LIN {X 0,Y 235.109,Z 274.18,A -85,B 0,C 180,E1 -19787.924,E2 -19787.924} C_VEL
LIN {X 0,Y 235.327,Z 274.163,A -85,B 0,C 180,E1 -19791.414,E2 -19791.414} C_VEL
LIN {X 0,Y 235.369,Z 274.162,A -85,B 0,C 180,E1 -19793.142,E2 -19793.142} C_VEL
LIN {X 0,Y 235.592,Z 274.14,A -85,B 0,C 180,E1 -19798.293,E2 -19798.293} C_VEL
LIN {X 0,Y 235.593,Z 274.134,A -85,B 0,C 180,E1 -19801.711,E2 -19801.711} C_VEL
LIN {X 0,Y 235.402,Z 274.153,A -85,B 0,C 180,E1 -19806.861,E2 -19806.861} C_VEL
LIN {X 0,Y 235.237,Z 274.182,A -85,B 0,C 180,E1 -19810.328,E2 -19810.328} C_VEL
LIN {X 0,Y 235.107,Z 274.198,A -85,B 0,C 180,E1 -19815.609,E2 -19815.609} C_VEL
LIN {X 0,Y 235.007,Z 274.203,A -85,B 0,C 180,E1 -19819.208,E2 -19819.208} C_VEL
LIN {X 0,Y 234.961,Z 274.215,A -85,B 0,C 180,E1 -19822.885,E2 -19822.885} C_VEL
LIN {X 0,Y 234.97,Z 274.212,A -85,B 0,C 180,E1 -19826.659,E2 -19826.659} C_VEL
LIN {X 0,Y 234.933,Z 274.22,A -85,B 0,C 180,E1 -19830.57,E2 -19830.57} C_VEL
LIN {X 0,Y 234.929,Z 274.22,A -85,B 0,C 180,E1 -19834.64,E2 -19834.64} C_VEL
LIN {X 0,Y 234.945,Z 274.221,A -85,B 0,C 180,E1 -19838.946,E2 -19838.946} C_VEL
LIN {X 0,Y 234.971,Z 274.365,A -85,B 0,C 180,E1 -19843.971,E2 -19843.971} C_VEL
LIN {X 0,Y 235.687,Z 278.299,A -85,B 0,C 180,E1 -19848.203,E2 -19848.203} C_VEL
LIN {X 0,Y 236.227,Z 281.355,A -85,B 0,C 180,E1 -19851.335,E2 -19851.335} C_VEL
LIN {X 0,Y 236.327,Z 282.58,A -85,B 0,C 180,E1 -19852.548,E2 -19852.548} C_VEL
LIN {X 0,Y 235.561,Z 284.082,A -85,B 0,C 180,E1 -19853.919,E2 -19853.919} C_VEL
LIN {X 0,Y 233.781,Z 285.659,A -85,B 0,C 180,E1 -19855.25,E2 -19855.25} C_VEL
LIN {X 0,Y 229.483,Z 288.871,A -85,B 0,C 180,E1 -19857.918,E2 -19857.918} C_VEL
LIN {X 0,Y 228.112,Z 290.471,A -85,B 0,C 180,E1 -19859.328,E2 -19859.328} C_VEL
LIN {X 0,Y 227.922,Z 290.995,A -85,B 0,C 180,E1 -19859.811,E2 -19859.811} C_VEL
LIN {X 0,Y 227.643,Z 292.579,A -85,B 0,C 180,E1 -19861.29,E2 -19861.29} C_VEL
LIN {X 0,Y 230.37,Z 306.658,A -85,B 0,C 180,E1 -19862.479,E2 -19862.479} C_VEL
LIN {X 0,Y 232.357,Z 320.143,A -85,B 0,C 180,E1 -19863.933,E2 -19863.933} C_VEL
LIN {X 0,Y 233.562,Z 332.37,A -85,B 0,C 180,E1 -19865.56,E2 -19865.56} C_VEL
LIN {X 0,Y 234.118,Z 342.965,A -85,B 0,C 180,E1 -19867.264,E2 -19867.264} C_VEL
LIN {X 0,Y 232.286,Z 353.457,A -85,B 0,C 180,E1 -19869.176,E2 -19869.176} C_VEL
LIN {X 0,Y 230.426,Z 363.523,A -85,B 0,C 180,E1 -19871.471,E2 -19871.471} C_VEL
LIN {X 0,Y 228.848,Z 372.161,A -85,B 0,C 180,E1 -19873.955,E2 -19873.955} C_VEL
LIN {X 0,Y 227.39,Z 379.539,A -85,B 0,C 180,E1 -19876.597,E2 -19876.597} C_VEL
LIN {X 0,Y 226.524,Z 385.469,A -85,B 0,C 180,E1 -19879.272,E2 -19879.272} C_VEL
LIN {X 0,Y 225.961,Z 390.122,A -85,B 0,C 180,E1 -19881.954,E2 -19881.954} C_VEL
LIN {X 0,Y 225.657,Z 393.634,A -85,B 0,C 180,E1 -19884.639,E2 -19884.639} C_VEL
LIN {X 0,Y 225.627,Z 395.395,A -85,B 0,C 180,E1 -19886.428,E2 -19886.428} C_VEL
LIN {X 0,Y 225.692,Z 396.715,A -85,B 0,C 180,E1 -19888.215,E2 -19888.215} C_VEL
LIN {X 0,Y 225.758,Z 397.627,A -85,B 0,C 180,E1 -19890,E2 -19890} C_VEL
LIN {X 0,Y 225.659,Z 398.135,A -85,B 0,C 180,E1 -19891.784,E2 -19891.784} C_VEL
LIN {X 0,Y 225.601,Z 398.096,A -85,B 0,C 180,E1 -19894.512,E2 -19894.512} C_VEL
LIN {X 0,Y 225.831,Z 397.183,A -85,B 0,C 180,E1 -19897.15,E2 -19897.15} C_VEL
LIN {X 0,Y 226.166,Z 396.101,A -85,B 0,C 180,E1 -19898.938,E2 -19898.938} C_VEL
LIN {X 0,Y 226.673,Z 394.603,A -85,B 0,C 180,E1 -19900.721,E2 -19900.721} C_VEL
LIN {X 0,Y 227.781,Z 391.576,A -85,B 0,C 180,E1 -19903.379,E2 -19903.379} C_VEL
LIN {X 0,Y 229.362,Z 387.538,A -85,B 0,C 180,E1 -19906.008,E2 -19906.008} C_VEL
LIN {X 0,Y 231.967,Z 381.395,A -85,B 0,C 180,E1 -19909.007,E2 -19909.007} C_VEL
LIN {X 0,Y 234.464,Z 374.434,A -85,B 0,C 180,E1 -19911.683,E2 -19911.683} C_VEL
LIN {X 0,Y 237.395,Z 366.72,A -85,B 0,C 180,E1 -19914.02,E2 -19914.02} C_VEL
LIN {X 0,Y 240.409,Z 358.529,A -85,B 0,C 180,E1 -19916.007,E2 -19916.007} C_VEL
LIN {X 0,Y 242.378,Z 352.8,A -85,B 0,C 180,E1 -19917.173,E2 -19917.173} C_VEL
LIN {X 0,Y 243.214,Z 343.096,A -85,B 0,C 180,E1 -19919.215,E2 -19919.215} C_VEL
LIN {X 0,Y 242.953,Z 333.446,A -85,B 0,C 180,E1 -19921.135,E2 -19921.135} C_VEL
LIN {X 0,Y 241.554,Z 322.509,A -85,B 0,C 180,E1 -19923.227,E2 -19923.227} C_VEL
LIN {X 0,Y 238.999,Z 311.749,A -85,B 0,C 180,E1 -19925.301,E2 -19925.301} C_VEL
LIN {X 0,Y 235.898,Z 302.595,A -85,B 0,C 180,E1 -19927.162,E2 -19927.162} C_VEL
LIN {X 0,Y 234.604,Z 299.647,A -85,B 0,C 180,E1 -19927.81,E2 -19927.81} C_VEL
LIN {X 0,Y 232.641,Z 295.3,A -85,B 0,C 180,E1 -19928.793,E2 -19928.793} C_VEL
LIN {X 0,Y 230.868,Z 292.3,A -85,B 0,C 180,E1 -19929.608,E2 -19929.608} C_VEL
LIN {X 0,Y 230.247,Z 290.185,A -85,B 0,C 180,E1 -19930.007,E2 -19930.007} C_VEL
LIN {X 0,Y 230.039,Z 288.162,A -85,B 0,C 180,E1 -19932.839,E2 -19932.839} C_VEL
LIN {X 0,Y 229.659,Z 285.357,A -85,B 0,C 180,E1 -19937.259,E2 -19937.259} C_VEL
LIN {X 0,Y 229.411,Z 283.843,A -85,B 0,C 180,E1 -19939.983,E2 -19939.983} C_VEL
LIN {X 0,Y 229.062,Z 281.787,A -85,B 0,C 180,E1 -19944.339,E2 -19944.339} C_VEL
LIN {X 0,Y 228.798,Z 280.217,A -85,B 0,C 180,E1 -19948.519,E2 -19948.519} C_VEL
LIN {X 0,Y 228.652,Z 278.956,A -85,B 0,C 180,E1 -19953.042,E2 -19953.042} C_VEL
LIN {X 0,Y 228.5,Z 278.111,A -85,B 0,C 180,E1 -19958.339,E2 -19958.339} C_VEL
LIN {X 0,Y 228.515,Z 277.888,A -85,B 0,C 180,E1 -19962.437,E2 -19962.437} C_VEL
LIN {X 0,Y 228.587,Z 277.979,A -85,B 0,C 180,E1 -19965.759,E2 -19965.759} C_VEL
LIN {X 0,Y 228.79,Z 278.339,A -85,B 0,C 180,E1 -19969.407,E2 -19969.407} C_VEL
LIN {X 0,Y 228.966,Z 278.971,A -85,B 0,C 180,E1 -19972.946,E2 -19972.946} C_VEL
LIN {X 0,Y 229.425,Z 280.374,A -85,B 0,C 180,E1 -19978.243,E2 -19978.243} C_VEL
LIN {X 0,Y 229.645,Z 280.948,A -85,B 0,C 180,E1 -19979.998,E2 -19979.998} C_VEL
LIN {X 0,Y 229.49,Z 282.382,A -85,B 0,C 180,E1 -19983.509,E2 -19983.509} C_VEL
LIN {X 0,Y 229.473,Z 283.455,A -85,B 0,C 180,E1 -19985.876,E2 -19985.876} C_VEL
LIN {X 0,Y 230.504,Z 286.209,A -85,B 0,C 180,E1 -19986.453,E2 -19986.453} C_VEL
LIN {X 0,Y 232.638,Z 289.092,A -85,B 0,C 180,E1 -19987.388,E2 -19987.388} C_VEL
LIN {X 0,Y 234.347,Z 292.521,A -85,B 0,C 180,E1 -19988.256,E2 -19988.256} C_VEL
LIN {X 0,Y 238.089,Z 300.635,A -85,B 0,C 180,E1 -19990.199,E2 -19990.199} C_VEL
LIN {X 0,Y 241.76,Z 311.494,A -85,B 0,C 180,E1 -19992.608,E2 -19992.608} C_VEL
LIN {X 0,Y 243.899,Z 320.884,A -85,B 0,C 180,E1 -19994.602,E2 -19994.602} C_VEL
LIN {X 0,Y 245.093,Z 330.377,A -85,B 0,C 180,E1 -19996.661,E2 -19996.661} C_VEL
LIN {X 0,Y 245.285,Z 336.573,A -85,B 0,C 180,E1 -19998.035,E2 -19998.035} C_VEL
LIN {X 0,Y 242.242,Z 346.347,A -85,B 0,C 180,E1 -19999.929,E2 -19999.929} C_VEL
LIN {X 0,Y 239.08,Z 355.259,A -85,B 0,C 180,E1 -20002.077,E2 -20002.077} C_VEL
LIN {X 0,Y 235.802,Z 363.65,A -85,B 0,C 180,E1 -20004.66,E2 -20004.66} C_VEL
LIN {X 0,Y 233.456,Z 369.311,A -85,B 0,C 180,E1 -20006.841,E2 -20006.841} C_VEL
LIN {X 0,Y 231.392,Z 374.044,A -85,B 0,C 180,E1 -20009.073,E2 -20009.073} C_VEL
LIN {X 0,Y 229.708,Z 377.876,A -85,B 0,C 180,E1 -20011.338,E2 -20011.338} C_VEL
LIN {X 0,Y 227.769,Z 382.127,A -85,B 0,C 180,E1 -20014.809,E2 -20014.809} C_VEL
LIN {X 0,Y 226.387,Z 384.802,A -85,B 0,C 180,E1 -20018.378,E2 -20018.378} C_VEL
LIN {X 0,Y 225.615,Z 385.794,A -85,B 0,C 180,E1 -20021.618,E2 -20021.618} C_VEL
LIN {X 0,Y 225.292,Z 385.696,A -85,B 0,C 180,E1 -20024.154,E2 -20024.154} C_VEL
LIN {X 0,Y 225.213,Z 384.787,A -85,B 0,C 180,E1 -20026.645,E2 -20026.645} C_VEL
LIN {X 0,Y 225.305,Z 383.158,A -85,B 0,C 180,E1 -20029.077,E2 -20029.077} C_VEL
LIN {X 0,Y 225.669,Z 380.804,A -85,B 0,C 180,E1 -20031.476,E2 -20031.476} C_VEL
LIN {X 0,Y 226.183,Z 377.61,A -85,B 0,C 180,E1 -20033.885,E2 -20033.885} C_VEL
LIN {X 0,Y 226.991,Z 372.694,A -85,B 0,C 180,E1 -20036.712,E2 -20036.712} C_VEL
LIN {X 0,Y 228.158,Z 366.18,A -85,B 0,C 180,E1 -20039.592,E2 -20039.592} C_VEL
LIN {X 0,Y 229.753,Z 357.785,A -85,B 0,C 180,E1 -20042.504,E2 -20042.504} C_VEL
LIN {X 0,Y 231.376,Z 349.279,A -85,B 0,C 180,E1 -20044.834,E2 -20044.834} C_VEL
LIN {X 0,Y 233.076,Z 339.892,A -85,B 0,C 180,E1 -20046.922,E2 -20046.922} C_VEL
LIN {X 0,Y 234.817,Z 330.283,A -85,B 0,C 180,E1 -20048.654,E2 -20048.654} C_VEL
LIN {X 0,Y 235.628,Z 324.925,A -85,B 0,C 180,E1 -20049.485,E2 -20049.485} C_VEL
LIN {X 0,Y 234.384,Z 314.919,A -85,B 0,C 180,E1 -20051.017,E2 -20051.017} C_VEL
LIN {X 0,Y 232.292,Z 302.871,A -85,B 0,C 180,E1 -20052.582,E2 -20052.582} C_VEL
LIN {X 0,Y 229.337,Z 289.586,A -85,B 0,C 180,E1 -20053.991,E2 -20053.991} C_VEL
LIN {X 0,Y 227.152,Z 280.91,A -85,B 0,C 180,E1 -20054.753,E2 -20054.753} C_VEL
LIN {X 0,Y 227.624,Z 277.181,A -85,B 0,C 180,E1 -20059.325,E2 -20059.325} C_VEL
LIN {X 0,Y 228.142,Z 275.067,A -85,B 0,C 180,E1 -20062.032,E2 -20062.032} C_VEL
LIN {X 0,Y 228.544,Z 275.016,A -85,B 0,C 180,E1 -20068.238,E2 -20068.238} C_VEL
LIN {X 0,Y 228.548,Z 275.015,A -85,B 0,C 180,E1 -20071.762,E2 -20071.762} C_VEL
LIN {X 0,Y 228.349,Z 275.041,A -85,B 0,C 180,E1 -20077.072,E2 -20077.072} C_VEL
LIN {X 0,Y 228.163,Z 275.062,A -85,B 0,C 180,E1 -20080.65,E2 -20080.65} C_VEL
LIN {X 0,Y 228.049,Z 275.077,A -85,B 0,C 180,E1 -20086.103,E2 -20086.103} C_VEL
LIN {X 0,Y 227.946,Z 275.088,A -85,B 0,C 180,E1 -20089.825,E2 -20089.825} C_VEL
LIN {X 0,Y 227.917,Z 275.095,A -85,B 0,C 180,E1 -20093.632,E2 -20093.632} C_VEL
LIN {X 0,Y 227.871,Z 275.093,A -85,B 0,C 180,E1 -20097.557,E2 -20097.557} C_VEL
LIN {X 0,Y 227.861,Z 275.1,A -85,B 0,C 180,E1 -20101.623,E2 -20101.623} C_VEL
LIN {X 0,Y 227.893,Z 275.097,A -85,B 0,C 180,E1 -20105.869,E2 -20105.869} C_VEL
LIN {X 0,Y 227.896,Z 275.085,A -85,B 0,C 180,E1 -20110.361,E2 -20110.361} C_VEL
LIN {X 0,Y 227.912,Z 275.086,A -85,B 0,C 180,E1 -20114.831,E2 -20114.831} C_VEL
LIN {X 0,Y 227.919,Z 275.093,A -85,B 0,C 180,E1 -20117.735,E2 -20117.735} C_VEL
LIN {X 0,Y 227.864,Z 275.099,A -85,B 0,C 180,E1 -20121.916,E2 -20121.916} C_VEL
LIN {X 0,Y 227.883,Z 275.089,A -85,B 0,C 180,E1 -20126.375,E2 -20126.375} C_VEL
LIN {X 0,Y 227.913,Z 275.078,A -85,B 0,C 180,E1 -20130.44,E2 -20130.44} C_VEL
LIN {X 0,Y 227.923,Z 275.088,A -85,B 0,C 180,E1 -20134.428,E2 -20134.428} C_VEL
LIN {X 0,Y 227.957,Z 275.089,A -85,B 0,C 180,E1 -20138.289,E2 -20138.289} C_VEL
LIN {X 0,Y 228.03,Z 275.076,A -85,B 0,C 180,E1 -20142.828,E2 -20142.828} C_VEL
LIN {X 0,Y 228.067,Z 275.056,A -85,B 0,C 180,E1 -20147.545,E2 -20147.545} C_VEL
LIN {X 0,Y 228.263,Z 275.043,A -85,B 0,C 180,E1 -20151.147,E2 -20151.147} C_VEL
LIN {X 0,Y 228.32,Z 275.041,A -85,B 0,C 180,E1 -20152.93,E2 -20152.93} C_VEL
LIN {X 0,Y 228.551,Z 275.017,A -85,B 0,C 180,E1 -20158.24,E2 -20158.24} C_VEL
LIN {X 0,Y 228.552,Z 275.011,A -85,B 0,C 180,E1 -20161.764,E2 -20161.764} C_VEL
LIN {X 0,Y 228.353,Z 275.031,A -85,B 0,C 180,E1 -20167.074,E2 -20167.074} C_VEL
LIN {X 0,Y 228.162,Z 275.062,A -85,B 0,C 180,E1 -20170.652,E2 -20170.652} C_VEL
LIN {X 0,Y 228.053,Z 275.073,A -85,B 0,C 180,E1 -20176.104,E2 -20176.104} C_VEL
LIN {X 0,Y 227.942,Z 275.086,A -85,B 0,C 180,E1 -20179.828,E2 -20179.828} C_VEL
LIN {X 0,Y 227.915,Z 275.097,A -85,B 0,C 180,E1 -20183.635,E2 -20183.635} C_VEL
LIN {X 0,Y 227.886,Z 275.095,A -85,B 0,C 180,E1 -20187.557,E2 -20187.557} C_VEL
LIN {X 0,Y 227.872,Z 275.103,A -85,B 0,C 180,E1 -20191.624,E2 -20191.624} C_VEL
LIN {X 0,Y 227.882,Z 275.097,A -85,B 0,C 180,E1 -20195.874,E2 -20195.874} C_VEL
LIN {X 0,Y 227.829,Z 275.104,A -85,B 0,C 180,E1 -20200.378,E2 -20200.378} C_VEL
LIN {X 0,Y 227.93,Z 275.125,A -85,B 0,C 180,E1 -20203.626,E2 -20203.626} C_VEL
LIN {X 0,Y 228.53,Z 278.675,A -85,B 0,C 180,E1 -20207.57,E2 -20207.57} C_VEL
LIN {X 0,Y 229.161,Z 282.067,A -85,B 0,C 180,E1 -20211.17,E2 -20211.17} C_VEL
LIN {X 0,Y 229.294,Z 283.707,A -85,B 0,C 180,E1 -20212.839,E2 -20212.839} C_VEL
LIN {X 0,Y 229.191,Z 285.251,A -85,B 0,C 180,E1 -20214.365,E2 -20214.365} C_VEL
LIN {X 0,Y 228.258,Z 289.527,A -85,B 0,C 180,E1 -20218.438,E2 -20218.438} C_VEL
LIN {X 0,Y 227.922,Z 290.995,A -85,B 0,C 180,E1 -20219.811,E2 -20219.811} C_VEL
LIN {X 0,Y 227.69,Z 292.595,A -85,B 0,C 180,E1 -20220.522,E2 -20220.522} C_VEL
LIN {X 0,Y 227.27,Z 296.129,A -85,B 0,C 180,E1 -20221.199,E2 -20221.199} C_VEL
LIN {X 0,Y 226.616,Z 301.709,A -85,B 0,C 180,E1 -20221.731,E2 -20221.731} C_VEL
LIN {X 0,Y 225.166,Z 314.703,A -85,B 0,C 180,E1 -20222.738,E2 -20222.738} C_VEL
LIN {X 0,Y 225.343,Z 319.397,A -85,B 0,C 180,E1 -20223.261,E2 -20223.261} C_VEL
LIN {X 0,Y 226.472,Z 330.659,A -85,B 0,C 180,E1 -20224.786,E2 -20224.786} C_VEL
LIN {X 0,Y 227.246,Z 342.743,A -85,B 0,C 180,E1 -20226.777,E2 -20226.777} C_VEL
LIN {X 0,Y 225.411,Z 353.248,A -85,B 0,C 180,E1 -20228.749,E2 -20228.749} C_VEL
LIN {X 0,Y 223.533,Z 362.941,A -85,B 0,C 180,E1 -20231.011,E2 -20231.011} C_VEL
LIN {X 0,Y 221.938,Z 371.269,A -85,B 0,C 180,E1 -20233.441,E2 -20233.441} C_VEL
LIN {X 0,Y 220.454,Z 378.773,A -85,B 0,C 180,E1 -20236.167,E2 -20236.167} C_VEL
LIN {X 0,Y 219.512,Z 384.809,A -85,B 0,C 180,E1 -20238.925,E2 -20238.925} C_VEL
LIN {X 0,Y 218.904,Z 389.56,A -85,B 0,C 180,E1 -20241.693,E2 -20241.693} C_VEL
LIN {X 0,Y 218.581,Z 393.165,A -85,B 0,C 180,E1 -20244.465,E2 -20244.465} C_VEL
LIN {X 0,Y 218.527,Z 395.006,A -85,B 0,C 180,E1 -20246.312,E2 -20246.312} C_VEL
LIN {X 0,Y 218.606,Z 396.372,A -85,B 0,C 180,E1 -20248.157,E2 -20248.157} C_VEL
LIN {X 0,Y 218.671,Z 397.323,A -85,B 0,C 180,E1 -20250,E2 -20250} C_VEL
LIN {X 0,Y 218.574,Z 397.87,A -85,B 0,C 180,E1 -20251.842,E2 -20251.842} C_VEL
LIN {X 0,Y 218.519,Z 397.943,A -85,B 0,C 180,E1 -20254.403,E2 -20254.403} C_VEL
LIN {X 0,Y 218.77,Z 397.089,A -85,B 0,C 180,E1 -20257.383,E2 -20257.383} C_VEL
LIN {X 0,Y 219.681,Z 394.626,A -85,B 0,C 180,E1 -20261.066,E2 -20261.066} C_VEL
LIN {X 0,Y 220.853,Z 391.671,A -85,B 0,C 180,E1 -20263.807,E2 -20263.807} C_VEL
LIN {X 0,Y 222.561,Z 387.73,A -85,B 0,C 180,E1 -20266.51,E2 -20266.51} C_VEL
LIN {X 0,Y 224.863,Z 382.723,A -85,B 0,C 180,E1 -20269.157,E2 -20269.157} C_VEL
LIN {X 0,Y 227.306,Z 376.526,A -85,B 0,C 180,E1 -20271.778,E2 -20271.778} C_VEL
LIN {X 0,Y 230.379,Z 368.865,A -85,B 0,C 180,E1 -20274.319,E2 -20274.319} C_VEL
LIN {X 0,Y 233.424,Z 361.125,A -85,B 0,C 180,E1 -20276.365,E2 -20276.365} C_VEL
LIN {X 0,Y 236.129,Z 353.835,A -85,B 0,C 180,E1 -20277.954,E2 -20277.954} C_VEL
LIN {X 0,Y 237.12,Z 343.537,A -85,B 0,C 180,E1 -20280.255,E2 -20280.255} C_VEL
LIN {X 0,Y 237.032,Z 335.241,A -85,B 0,C 180,E1 -20282.004,E2 -20282.004} C_VEL
LIN {X 0,Y 235.875,Z 324.703,A -85,B 0,C 180,E1 -20284.157,E2 -20284.157} C_VEL
LIN {X 0,Y 233.34,Z 313.355,A -85,B 0,C 180,E1 -20286.523,E2 -20286.523} C_VEL
LIN {X 0,Y 230.672,Z 305.204,A -85,B 0,C 180,E1 -20288.319,E2 -20288.319} C_VEL
LIN {X 0,Y 228.334,Z 300.11,A -85,B 0,C 180,E1 -20289.624,E2 -20289.624} C_VEL
LIN {X 0,Y 226.59,Z 296.359,A -85,B 0,C 180,E1 -20290.586,E2 -20290.586} C_VEL
LIN {X 0,Y 223.827,Z 292.087,A -85,B 0,C 180,E1 -20291.976,E2 -20291.976} C_VEL
LIN {X 0,Y 223.131,Z 289.834,A -85,B 0,C 180,E1 -20292.466,E2 -20292.466} C_VEL
LIN {X 0,Y 222.765,Z 287.298,A -85,B 0,C 180,E1 -20296.519,E2 -20296.519} C_VEL
LIN {X 0,Y 222.404,Z 285.015,A -85,B 0,C 180,E1 -20300.8,E2 -20300.8} C_VEL
LIN {X 0,Y 222.282,Z 283.94,A -85,B 0,C 180,E1 -20303.075,E2 -20303.075} C_VEL
LIN {X 0,Y 221.909,Z 281.809,A -85,B 0,C 180,E1 -20308.769,E2 -20308.769} C_VEL
LIN {X 0,Y 221.73,Z 280.535,A -85,B 0,C 180,E1 -20313.655,E2 -20313.655} C_VEL
LIN {X 0,Y 221.621,Z 279.903,A -85,B 0,C 180,E1 -20317.631,E2 -20317.631} C_VEL
LIN {X 0,Y 221.618,Z 279.603,A -85,B 0,C 180,E1 -20322.054,E2 -20322.054} C_VEL
LIN {X 0,Y 221.742,Z 279.781,A -85,B 0,C 180,E1 -20327.18,E2 -20327.18} C_VEL
LIN {X 0,Y 221.981,Z 280.226,A -85,B 0,C 180,E1 -20330.89,E2 -20330.89} C_VEL
LIN {X 0,Y 222.095,Z 280.973,A -85,B 0,C 180,E1 -20334.55,E2 -20334.55} C_VEL
LIN {X 0,Y 222.483,Z 281.915,A -85,B 0,C 180,E1 -20338.188,E2 -20338.188} C_VEL
LIN {X 0,Y 222.723,Z 282.485,A -85,B 0,C 180,E1 -20339.998,E2 -20339.998} C_VEL
LIN {X 0,Y 222.565,Z 283.867,A -85,B 0,C 180,E1 -20343.449,E2 -20343.449} C_VEL
LIN {X 0,Y 223.585,Z 286.659,A -85,B 0,C 180,E1 -20344.11,E2 -20344.11} C_VEL
LIN {X 0,Y 225.858,Z 289.561,A -85,B 0,C 180,E1 -20345.244,E2 -20345.244} C_VEL
LIN {X 0,Y 227.79,Z 293.241,A -85,B 0,C 180,E1 -20346.308,E2 -20346.308} C_VEL
LIN {X 0,Y 228.833,Z 294.901,A -85,B 0,C 180,E1 -20346.833,E2 -20346.833} C_VEL
LIN {X 0,Y 232.06,Z 301.788,A -85,B 0,C 180,E1 -20348.707,E2 -20348.707} C_VEL
LIN {X 0,Y 235.597,Z 311.998,A -85,B 0,C 180,E1 -20351.178,E2 -20351.178} C_VEL
LIN {X 0,Y 237.724,Z 321.242,A -85,B 0,C 180,E1 -20353.309,E2 -20353.309} C_VEL
LIN {X 0,Y 238.91,Z 330.177,A -85,B 0,C 180,E1 -20355.35,E2 -20355.35} C_VEL
LIN {X 0,Y 239.149,Z 337.532,A -85,B 0,C 180,E1 -20357.088,E2 -20357.088} C_VEL
LIN {X 0,Y 238.37,Z 340.868,A -85,B 0,C 180,E1 -20357.768,E2 -20357.768} C_VEL
LIN {X 0,Y 234.671,Z 351.265,A -85,B 0,C 180,E1 -20360.027,E2 -20360.027} C_VEL
LIN {X 0,Y 231.462,Z 359.483,A -85,B 0,C 180,E1 -20362.303,E2 -20362.303} C_VEL
LIN {X 0,Y 228.097,Z 367.313,A -85,B 0,C 180,E1 -20365.063,E2 -20365.063} C_VEL
LIN {X 0,Y 225.244,Z 373.544,A -85,B 0,C 180,E1 -20367.904,E2 -20367.904} C_VEL
LIN {X 0,Y 223.335,Z 377.492,A -85,B 0,C 180,E1 -20370.229,E2 -20370.229} C_VEL
LIN {X 0,Y 221.811,Z 380.64,A -85,B 0,C 180,E1 -20372.588,E2 -20372.588} C_VEL
LIN {X 0,Y 220.572,Z 383.083,A -85,B 0,C 180,E1 -20374.993,E2 -20374.993} C_VEL
LIN {X 0,Y 219.566,Z 384.776,A -85,B 0,C 180,E1 -20377.454,E2 -20377.454} C_VEL
LIN {X 0,Y 218.858,Z 385.772,A -85,B 0,C 180,E1 -20379.956,E2 -20379.956} C_VEL
LIN {X 0,Y 218.37,Z 386.06,A -85,B 0,C 180,E1 -20382.518,E2 -20382.518} C_VEL
LIN {X 0,Y 218.151,Z 385.546,A -85,B 0,C 180,E1 -20385.13,E2 -20385.13} C_VEL
LIN {X 0,Y 218.13,Z 384.183,A -85,B 0,C 180,E1 -20387.817,E2 -20387.817} C_VEL
LIN {X 0,Y 218.392,Z 381.901,A -85,B 0,C 180,E1 -20390.56,E2 -20390.56} C_VEL
LIN {X 0,Y 218.947,Z 378.567,A -85,B 0,C 180,E1 -20393.363,E2 -20393.363} C_VEL
LIN {X 0,Y 219.736,Z 373.943,A -85,B 0,C 180,E1 -20396.257,E2 -20396.257} C_VEL
LIN {X 0,Y 220.932,Z 367.358,A -85,B 0,C 180,E1 -20399.406,E2 -20399.406} C_VEL
LIN {X 0,Y 222.428,Z 359.779,A -85,B 0,C 180,E1 -20402.21,E2 -20402.21} C_VEL
LIN {X 0,Y 223.972,Z 351.723,A -85,B 0,C 180,E1 -20404.613,E2 -20404.613} C_VEL
LIN {X 0,Y 225.748,Z 342.461,A -85,B 0,C 180,E1 -20406.857,E2 -20406.857} C_VEL
LIN {X 0,Y 227.81,Z 331.358,A -85,B 0,C 180,E1 -20408.984,E2 -20408.984} C_VEL
LIN {X 0,Y 228.744,Z 324.991,A -85,B 0,C 180,E1 -20410.014,E2 -20410.014} C_VEL
LIN {X 0,Y 227.271,Z 313.977,A -85,B 0,C 180,E1 -20411.755,E2 -20411.755} C_VEL
LIN {X 0,Y 225.176,Z 302.364,A -85,B 0,C 180,E1 -20413.291,E2 -20413.291} C_VEL
LIN {X 0,Y 222.114,Z 288.88,A -85,B 0,C 180,E1 -20414.751,E2 -20414.751} C_VEL
LIN {X 0,Y 220.157,Z 281.048,A -85,B 0,C 180,E1 -20415.5,E2 -20415.5} C_VEL
LIN {X 0,Y 221.033,Z 276.124,A -85,B 0,C 180,E1 -20421.774,E2 -20421.774} C_VEL
LIN {X 0,Y 221.091,Z 275.944,A -85,B 0,C 180,E1 -20424.528,E2 -20424.528} C_VEL
LIN {X 0,Y 221.501,Z 275.893,A -85,B 0,C 180,E1 -20428.182,E2 -20428.182} C_VEL
LIN {X 0,Y 221.506,Z 275.892,A -85,B 0,C 180,E1 -20431.818,E2 -20431.818} C_VEL
LIN {X 0,Y 221.302,Z 275.919,A -85,B 0,C 180,E1 -20437.298,E2 -20437.298} C_VEL
LIN {X 0,Y 221.108,Z 275.939,A -85,B 0,C 180,E1 -20440.994,E2 -20440.994} C_VEL
LIN {X 0,Y 221.008,Z 275.951,A -85,B 0,C 180,E1 -20446.63,E2 -20446.63} C_VEL
LIN {X 0,Y 220.901,Z 275.968,A -85,B 0,C 180,E1 -20450.485,E2 -20450.485} C_VEL
LIN {X 0,Y 220.865,Z 275.97,A -85,B 0,C 180,E1 -20454.435,E2 -20454.435} C_VEL
LIN {X 0,Y 220.818,Z 275.969,A -85,B 0,C 180,E1 -20458.516,E2 -20458.516} C_VEL
LIN {X 0,Y 220.815,Z 275.977,A -85,B 0,C 180,E1 -20462.756,E2 -20462.756} C_VEL
LIN {X 0,Y 220.83,Z 275.976,A -85,B 0,C 180,E1 -20467.289,E2 -20467.289} C_VEL
LIN {X 0,Y 220.866,Z 275.957,A -85,B 0,C 180,E1 -20471.93,E2 -20471.93} C_VEL
LIN {X 0,Y 220.866,Z 275.969,A -85,B 0,C 180,E1 -20475.573,E2 -20475.573} C_VEL
LIN {X 0,Y 220.851,Z 275.974,A -85,B 0,C 180,E1 -20479.794,E2 -20479.794} C_VEL
LIN {X 0,Y 220.828,Z 275.976,A -85,B 0,C 180,E1 -20482.797,E2 -20482.797} C_VEL
LIN {X 0,Y 220.817,Z 275.964,A -85,B 0,C 180,E1 -20487.247,E2 -20487.247} C_VEL
LIN {X 0,Y 220.83,Z 275.966,A -85,B 0,C 180,E1 -20491.488,E2 -20491.488} C_VEL
LIN {X 0,Y 220.862,Z 275.97,A -85,B 0,C 180,E1 -20495.567,E2 -20495.567} C_VEL
LIN {X 0,Y 220.887,Z 275.968,A -85,B 0,C 180,E1 -20499.516,E2 -20499.516} C_VEL
LIN {X 0,Y 221.011,Z 275.947,A -85,B 0,C 180,E1 -20503.372,E2 -20503.372} C_VEL
LIN {X 0,Y 221.063,Z 275.933,A -85,B 0,C 180,E1 -20509.006,E2 -20509.006} C_VEL
LIN {X 0,Y 221.255,Z 275.922,A -85,B 0,C 180,E1 -20512.703,E2 -20512.703} C_VEL
LIN {X 0,Y 221.509,Z 275.894,A -85,B 0,C 180,E1 -20518.184,E2 -20518.184} C_VEL
LIN {X 0,Y 221.51,Z 275.888,A -85,B 0,C 180,E1 -20521.82,E2 -20521.82} C_VEL
LIN {X 0,Y 221.288,Z 275.911,A -85,B 0,C 180,E1 -20527.301,E2 -20527.301} C_VEL
LIN {X 0,Y 221.111,Z 275.94,A -85,B 0,C 180,E1 -20530.996,E2 -20530.996} C_VEL
LIN {X 0,Y 221.014,Z 275.947,A -85,B 0,C 180,E1 -20536.632,E2 -20536.632} C_VEL
LIN {X 0,Y 220.892,Z 275.965,A -85,B 0,C 180,E1 -20540.488,E2 -20540.488} C_VEL
LIN {X 0,Y 220.868,Z 275.971,A -85,B 0,C 180,E1 -20544.437,E2 -20544.437} C_VEL
LIN {X 0,Y 220.837,Z 275.971,A -85,B 0,C 180,E1 -20548.516,E2 -20548.516} C_VEL
LIN {X 0,Y 220.819,Z 275.98,A -85,B 0,C 180,E1 -20552.758,E2 -20552.758} C_VEL
LIN {X 0,Y 220.813,Z 275.981,A -85,B 0,C 180,E1 -20557.28,E2 -20557.28} C_VEL
LIN {X 0,Y 220.794,Z 275.982,A -85,B 0,C 180,E1 -20561.949,E2 -20561.949} C_VEL
LIN {X 0,Y 220.912,Z 276.165,A -85,B 0,C 180,E1 -20563.598,E2 -20563.598} C_VEL
LIN {X 0,Y 221.599,Z 280.249,A -85,B 0,C 180,E1 -20568.24,E2 -20568.24} C_VEL
LIN {X 0,Y 222.24,Z 283.946,A -85,B 0,C 180,E1 -20572.243,E2 -20572.243} C_VEL
LIN {X 0,Y 221.88,Z 287.103,A -85,B 0,C 180,E1 -20575.444,E2 -20575.444} C_VEL
LIN {X 0,Y 220.86,Z 291.459,A -85,B 0,C 180,E1 -20579.678,E2 -20579.678} C_VEL
LIN {X 0,Y 220.702,Z 292.38,A -85,B 0,C 180,E1 -20580.568,E2 -20580.568} C_VEL
LIN {X 0,Y 223.474,Z 306.806,A -85,B 0,C 180,E1 -20581.853,E2 -20581.853} C_VEL
LIN {X 0,Y 225.343,Z 319.397,A -85,B 0,C 180,E1 -20583.261,E2 -20583.261} C_VEL
LIN {X 0,Y 225.432,Z 324.737,A -85,B 0,C 180,E1 -20583.903,E2 -20583.903} C_VEL
LIN {X 0,Y 224.576,Z 330.049,A -85,B 0,C 180,E1 -20584.541,E2 -20584.541} C_VEL
LIN {X 0,Y 221.541,Z 340.322,A -85,B 0,C 180,E1 -20585.93,E2 -20585.93} C_VEL
LIN {X 0,Y 219.753,Z 346.849,A -85,B 0,C 180,E1 -20587.048,E2 -20587.048} C_VEL
LIN {X 0,Y 217.718,Z 357.051,A -85,B 0,C 180,E1 -20589.202,E2 -20589.202} C_VEL
LIN {X 0,Y 216.071,Z 365.841,A -85,B 0,C 180,E1 -20591.51,E2 -20591.51} C_VEL
LIN {X 0,Y 214.573,Z 373.089,A -85,B 0,C 180,E1 -20593.835,E2 -20593.835} C_VEL
LIN {X 0,Y 213.093,Z 380.206,A -85,B 0,C 180,E1 -20596.652,E2 -20596.652} C_VEL
LIN {X 0,Y 212.268,Z 385.891,A -85,B 0,C 180,E1 -20599.508,E2 -20599.508} C_VEL
LIN {X 0,Y 211.714,Z 390.338,A -85,B 0,C 180,E1 -20602.369,E2 -20602.369} C_VEL
LIN {X 0,Y 211.431,Z 394.148,A -85,B 0,C 180,E1 -20605.74,E2 -20605.74} C_VEL
LIN {X 0,Y 211.503,Z 396.01,A -85,B 0,C 180,E1 -20608.096,E2 -20608.096} C_VEL
LIN {X 0,Y 211.585,Z 397.007,A -85,B 0,C 180,E1 -20610,E2 -20610} C_VEL
LIN {X 0,Y 211.473,Z 397.598,A -85,B 0,C 180,E1 -20611.904,E2 -20611.904} C_VEL
LIN {X 0,Y 211.425,Z 397.796,A -85,B 0,C 180,E1 -20614.241,E2 -20614.241} C_VEL
LIN {X 0,Y 211.701,Z 396.995,A -85,B 0,C 180,E1 -20617.63,E2 -20617.63} C_VEL
LIN {X 0,Y 212.705,Z 394.626,A -85,B 0,C 180,E1 -20621.434,E2 -20621.434} C_VEL
LIN {X 0,Y 213.945,Z 391.783,A -85,B 0,C 180,E1 -20624.262,E2 -20624.262} C_VEL
LIN {X 0,Y 215.778,Z 387.961,A -85,B 0,C 180,E1 -20627.045,E2 -20627.045} C_VEL
LIN {X 0,Y 218.178,Z 383.069,A -85,B 0,C 180,E1 -20629.768,E2 -20629.768} C_VEL
LIN {X 0,Y 221.185,Z 375.996,A -85,B 0,C 180,E1 -20632.856,E2 -20632.856} C_VEL
LIN {X 0,Y 224.586,Z 368.117,A -85,B 0,C 180,E1 -20635.485,E2 -20635.485} C_VEL
LIN {X 0,Y 228.513,Z 358.597,A -85,B 0,C 180,E1 -20637.97,E2 -20637.97} C_VEL
LIN {X 0,Y 229.919,Z 354.92,A -85,B 0,C 180,E1 -20638.778,E2 -20638.778} C_VEL
LIN {X 0,Y 231.011,Z 345.841,A -85,B 0,C 180,E1 -20640.931,E2 -20640.931} C_VEL
LIN {X 0,Y 231.079,Z 336.939,A -85,B 0,C 180,E1 -20642.931,E2 -20642.931} C_VEL
LIN {X 0,Y 230.137,Z 326.538,A -85,B 0,C 180,E1 -20645.221,E2 -20645.221} C_VEL
LIN {X 0,Y 227.961,Z 316.091,A -85,B 0,C 180,E1 -20647.576,E2 -20647.576} C_VEL
LIN {X 0,Y 226.208,Z 309.918,A -85,B 0,C 180,E1 -20649.036,E2 -20649.036} C_VEL
LIN {X 0,Y 223.881,Z 304.579,A -85,B 0,C 180,E1 -20650.511,E2 -20650.511} C_VEL
LIN {X 0,Y 222.182,Z 300.771,A -85,B 0,C 180,E1 -20651.594,E2 -20651.594} C_VEL
LIN {X 0,Y 220.134,Z 297.271,A -85,B 0,C 180,E1 -20652.796,E2 -20652.796} C_VEL
LIN {X 0,Y 219.291,Z 295.337,A -85,B 0,C 180,E1 -20653.338,E2 -20653.338} C_VEL
LIN {X 0,Y 216.81,Z 292.113,A -85,B 0,C 180,E1 -20654.72,E2 -20654.72} C_VEL
LIN {X 0,Y 215.878,Z 289.432,A -85,B 0,C 180,E1 -20655.427,E2 -20655.427} C_VEL
LIN {X 0,Y 215.587,Z 287.315,A -85,B 0,C 180,E1 -20659.306,E2 -20659.306} C_VEL
LIN {X 0,Y 215.44,Z 286.174,A -85,B 0,C 180,E1 -20661.695,E2 -20661.695} C_VEL
LIN {X 0,Y 215.085,Z 284.334,A -85,B 0,C 180,E1 -20666.254,E2 -20666.254} C_VEL
LIN {X 0,Y 215.028,Z 283.579,A -85,B 0,C 180,E1 -20668.468,E2 -20668.468} C_VEL
LIN {X 0,Y 214.883,Z 282.438,A -85,B 0,C 180,E1 -20672.747,E2 -20672.747} C_VEL
LIN {X 0,Y 214.744,Z 281.725,A -85,B 0,C 180,E1 -20676.873,E2 -20676.873} C_VEL
LIN {X 0,Y 214.702,Z 281.338,A -85,B 0,C 180,E1 -20681.669,E2 -20681.669} C_VEL
LIN {X 0,Y 214.779,Z 281.339,A -85,B 0,C 180,E1 -20684.822,E2 -20684.822} C_VEL
LIN {X 0,Y 214.926,Z 281.626,A -85,B 0,C 180,E1 -20688.803,E2 -20688.803} C_VEL
LIN {X 0,Y 215.124,Z 282.163,A -85,B 0,C 180,E1 -20692.489,E2 -20692.489} C_VEL
LIN {X 0,Y 215.572,Z 283.473,A -85,B 0,C 180,E1 -20698.13,E2 -20698.13} C_VEL
LIN {X 0,Y 215.778,Z 284.396,A -85,B 0,C 180,E1 -20700.639,E2 -20700.639} C_VEL
LIN {X 0,Y 216.765,Z 287.027,A -85,B 0,C 180,E1 -20701.391,E2 -20701.391} C_VEL
LIN {X 0,Y 219.242,Z 290.202,A -85,B 0,C 180,E1 -20702.82,E2 -20702.82} C_VEL
LIN {X 0,Y 220.965,Z 293.598,A -85,B 0,C 180,E1 -20703.93,E2 -20703.93} C_VEL
LIN {X 0,Y 222.097,Z 294.979,A -85,B 0,C 180,E1 -20704.535,E2 -20704.535} C_VEL
LIN {X 0,Y 226.212,Z 303.282,A -85,B 0,C 180,E1 -20707.137,E2 -20707.137} C_VEL
LIN {X 0,Y 229.069,Z 311.366,A -85,B 0,C 180,E1 -20709.308,E2 -20709.308} C_VEL
LIN {X 0,Y 231.247,Z 319.549,A -85,B 0,C 180,E1 -20711.391,E2 -20711.391} C_VEL
LIN {X 0,Y 232.616,Z 328.271,A -85,B 0,C 180,E1 -20713.539,E2 -20713.539} C_VEL
LIN {X 0,Y 233.083,Z 337.204,A -85,B 0,C 180,E1 -20715.744,E2 -20715.744} C_VEL
LIN {X 0,Y 233.037,Z 339.907,A -85,B 0,C 180,E1 -20716.421,E2 -20716.421} C_VEL
LIN {X 0,Y 229.689,Z 349.353,A -85,B 0,C 180,E1 -20718.466,E2 -20718.466} C_VEL
LIN {X 0,Y 226.652,Z 356.822,A -85,B 0,C 180,E1 -20720.437,E2 -20720.437} C_VEL
LIN {X 0,Y 222.918,Z 365.254,A -85,B 0,C 180,E1 -20723.237,E2 -20723.237} C_VEL
LIN {X 0,Y 219.496,Z 372.314,A -85,B 0,C 180,E1 -20726.298,E2 -20726.298} C_VEL
LIN {X 0,Y 217.064,Z 377.14,A -85,B 0,C 180,E1 -20729.053,E2 -20729.053} C_VEL
LIN {X 0,Y 215.099,Z 380.844,A -85,B 0,C 180,E1 -20731.844,E2 -20731.844} C_VEL
LIN {X 0,Y 213.595,Z 383.534,A -85,B 0,C 180,E1 -20734.658,E2 -20734.658} C_VEL
LIN {X 0,Y 212.469,Z 385.286,A -85,B 0,C 180,E1 -20737.454,E2 -20737.454} C_VEL
LIN {X 0,Y 211.685,Z 386.148,A -85,B 0,C 180,E1 -20740.219,E2 -20740.219} C_VEL
LIN {X 0,Y 211.206,Z 386.182,A -85,B 0,C 180,E1 -20742.942,E2 -20742.942} C_VEL
LIN {X 0,Y 211.03,Z 385.445,A -85,B 0,C 180,E1 -20745.625,E2 -20745.625} C_VEL
LIN {X 0,Y 211.041,Z 383.984,A -85,B 0,C 180,E1 -20748.24,E2 -20748.24} C_VEL
LIN {X 0,Y 211.54,Z 380.579,A -85,B 0,C 180,E1 -20751.887,E2 -20751.887} C_VEL
LIN {X 0,Y 212.138,Z 377.032,A -85,B 0,C 180,E1 -20754.567,E2 -20754.567} C_VEL
LIN {X 0,Y 213.045,Z 371.818,A -85,B 0,C 180,E1 -20757.585,E2 -20757.585} C_VEL
LIN {X 0,Y 214.309,Z 365.29,A -85,B 0,C 180,E1 -20760.535,E2 -20760.535} C_VEL
LIN {X 0,Y 215.981,Z 357.152,A -85,B 0,C 180,E1 -20763.423,E2 -20763.423} C_VEL
LIN {X 0,Y 217.803,Z 348.179,A -85,B 0,C 180,E1 -20765.96,E2 -20765.96} C_VEL
LIN {X 0,Y 219.747,Z 338.175,A -85,B 0,C 180,E1 -20768.238,E2 -20768.238} C_VEL
LIN {X 0,Y 221.831,Z 326.462,A -85,B 0,C 180,E1 -20770.33,E2 -20770.33} C_VEL
LIN {X 0,Y 220.511,Z 315.525,A -85,B 0,C 180,E1 -20772.136,E2 -20772.136} C_VEL
LIN {X 0,Y 218.636,Z 304.682,A -85,B 0,C 180,E1 -20773.665,E2 -20773.665} C_VEL
LIN {X 0,Y 215.759,Z 291.589,A -85,B 0,C 180,E1 -20775.198,E2 -20775.198} C_VEL
LIN {X 0,Y 213.14,Z 281.255,A -85,B 0,C 180,E1 -20776.23,E2 -20776.23} C_VEL
LIN {X 0,Y 214.042,Z 276.822,A -85,B 0,C 180,E1 -20782.12,E2 -20782.12} C_VEL
LIN {X 0,Y 214.434,Z 276.773,A -85,B 0,C 180,E1 -20788.122,E2 -20788.122} C_VEL
LIN {X 0,Y 214.545,Z 276.759,A -85,B 0,C 180,E1 -20790,E2 -20790} C_VEL
LIN {X 0,Y 214.439,Z 276.773,A -85,B 0,C 180,E1 -20791.878,E2 -20791.878} C_VEL
LIN {X 0,Y 214.239,Z 276.799,A -85,B 0,C 180,E1 -20797.54,E2 -20797.54} C_VEL
LIN {X 0,Y 214.039,Z 276.82,A -85,B 0,C 180,E1 -20801.362,E2 -20801.362} C_VEL
LIN {X 0,Y 213.925,Z 276.836,A -85,B 0,C 180,E1 -20805.237,E2 -20805.237} C_VEL
LIN {X 0,Y 213.868,Z 276.839,A -85,B 0,C 180,E1 -20809.185,E2 -20809.185} C_VEL
LIN {X 0,Y 213.848,Z 276.846,A -85,B 0,C 180,E1 -20813.227,E2 -20813.227} C_VEL
LIN {X 0,Y 213.82,Z 276.842,A -85,B 0,C 180,E1 -20817.451,E2 -20817.451} C_VEL
LIN {X 0,Y 213.761,Z 276.857,A -85,B 0,C 180,E1 -20821.738,E2 -20821.738} C_VEL
LIN {X 0,Y 213.747,Z 276.857,A -85,B 0,C 180,E1 -20826.287,E2 -20826.287} C_VEL
LIN {X 0,Y 213.816,Z 276.837,A -85,B 0,C 180,E1 -20831.1,E2 -20831.1} C_VEL
LIN {X 0,Y 213.829,Z 276.838,A -85,B 0,C 180,E1 -20833.694,E2 -20833.694} C_VEL
LIN {X 0,Y 213.833,Z 276.844,A -85,B 0,C 180,E1 -20836.358,E2 -20836.358} C_VEL
LIN {X 0,Y 213.814,Z 276.851,A -85,B 0,C 180,E1 -20839.112,E2 -20839.112} C_VEL
LIN {X 0,Y 213.747,Z 276.854,A -85,B 0,C 180,E1 -20843.716,E2 -20843.716} C_VEL
LIN {X 0,Y 213.79,Z 276.835,A -85,B 0,C 180,E1 -20848.726,E2 -20848.726} C_VEL
LIN {X 0,Y 213.82,Z 276.84,A -85,B 0,C 180,E1 -20852.605,E2 -20852.605} C_VEL
LIN {X 0,Y 213.847,Z 276.848,A -85,B 0,C 180,E1 -20856.955,E2 -20856.955} C_VEL
LIN {X 0,Y 213.939,Z 276.83,A -85,B 0,C 180,E1 -20862.806,E2 -20862.806} C_VEL
LIN {X 0,Y 213.947,Z 276.815,A -85,B 0,C 180,E1 -20866.709,E2 -20866.709} C_VEL
LIN {X 0,Y 214.138,Z 276.799,A -85,B 0,C 180,E1 -20870.557,E2 -20870.557} C_VEL
LIN {X 0,Y 214.097,Z 276.815,A -85,B 0,C 180,E1 -20874.351,E2 -20874.351} C_VEL
LIN {X 0,Y 214.442,Z 276.774,A -85,B 0,C 180,E1 -20878.124,E2 -20878.124} C_VEL
LIN {X 0,Y 214.547,Z 276.759,A -85,B 0,C 180,E1 -20880.002,E2 -20880.002} C_VEL
LIN {X 0,Y 214.443,Z 276.767,A -85,B 0,C 180,E1 -20881.88,E2 -20881.88} C_VEL
LIN {X 0,Y 214.226,Z 276.79,A -85,B 0,C 180,E1 -20887.543,E2 -20887.543} C_VEL
LIN {X 0,Y 214.044,Z 276.821,A -85,B 0,C 180,E1 -20891.364,E2 -20891.364} C_VEL
LIN {X 0,Y 213.93,Z 276.834,A -85,B 0,C 180,E1 -20895.239,E2 -20895.239} C_VEL
LIN {X 0,Y 213.839,Z 276.838,A -85,B 0,C 180,E1 -20899.19,E2 -20899.19} C_VEL
LIN {X 0,Y 213.848,Z 276.846,A -85,B 0,C 180,E1 -20903.229,E2 -20903.229} C_VEL
LIN {X 0,Y 213.831,Z 276.845,A -85,B 0,C 180,E1 -20907.452,E2 -20907.452} C_VEL
LIN {X 0,Y 213.77,Z 276.859,A -85,B 0,C 180,E1 -20911.739,E2 -20911.739} C_VEL
LIN {X 0,Y 213.746,Z 276.857,A -85,B 0,C 180,E1 -20916.29,E2 -20916.29} C_VEL
LIN {X 0,Y 213.726,Z 276.863,A -85,B 0,C 180,E1 -20921.125,E2 -20921.125} C_VEL
LIN {X 0,Y 213.872,Z 276.98,A -85,B 0,C 180,E1 -20923.314,E2 -20923.314} C_VEL
LIN {X 0,Y 214.482,Z 280.755,A -85,B 0,C 180,E1 -20927.757,E2 -20927.757} C_VEL
LIN {X 0,Y 215.093,Z 284.216,A -85,B 0,C 180,E1 -20931.648,E2 -20931.648} C_VEL
LIN {X 0,Y 215.098,Z 286.395,A -85,B 0,C 180,E1 -20933.977,E2 -20933.977} C_VEL
LIN {X 0,Y 214.03,Z 290.982,A -85,B 0,C 180,E1 -20938.625,E2 -20938.625} C_VEL
LIN {X 0,Y 213.739,Z 292.234,A -85,B 0,C 180,E1 -20939.877,E2 -20939.877} C_VEL
LIN {X 0,Y 216.255,Z 305.461,A -85,B 0,C 180,E1 -20941.05,E2 -20941.05} C_VEL
LIN {X 0,Y 218.219,Z 317.828,A -85,B 0,C 180,E1 -20942.461,E2 -20942.461} C_VEL
LIN {X 0,Y 219.457,Z 329.481,A -85,B 0,C 180,E1 -20944.061,E2 -20944.061} C_VEL
LIN {X 0,Y 220.263,Z 341.151,A -85,B 0,C 180,E1 -20945.995,E2 -20945.995} C_VEL
LIN {X 0,Y 220.108,Z 345.107,A -85,B 0,C 180,E1 -20946.726,E2 -20946.726} C_VEL
LIN {X 0,Y 219.753,Z 346.849,A -85,B 0,C 180,E1 -20947.048,E2 -20947.048} C_VEL
LIN {X 0,Y 218.44,Z 349.989,A -85,B 0,C 180,E1 -20947.611,E2 -20947.611} C_VEL
LIN {X 0,Y 210.871,Z 359.104,A -85,B 0,C 180,E1 -20949.363,E2 -20949.363} C_VEL
LIN {X 0,Y 209.729,Z 361.847,A -85,B 0,C 180,E1 -20950.068,E2 -20950.068} C_VEL
LIN {X 0,Y 208.236,Z 369.317,A -85,B 0,C 180,E1 -20952.317,E2 -20952.317} C_VEL
LIN {X 0,Y 206.604,Z 377.145,A -85,B 0,C 180,E1 -20955.219,E2 -20955.219} C_VEL
LIN {X 0,Y 205.496,Z 383.404,A -85,B 0,C 180,E1 -20958.159,E2 -20958.159} C_VEL
LIN {X 0,Y 204.838,Z 388.368,A -85,B 0,C 180,E1 -20961.118,E2 -20961.118} C_VEL
LIN {X 0,Y 204.445,Z 392.166,A -85,B 0,C 180,E1 -20964.081,E2 -20964.081} C_VEL
LIN {X 0,Y 204.345,Z 394.109,A -85,B 0,C 180,E1 -20966.056,E2 -20966.056} C_VEL
LIN {X 0,Y 204.403,Z 395.63,A -85,B 0,C 180,E1 -20968.029,E2 -20968.029} C_VEL
LIN {X 0,Y 204.502,Z 396.691,A -85,B 0,C 180,E1 -20970,E2 -20970} C_VEL
LIN {X 0,Y 204.374,Z 397.326,A -85,B 0,C 180,E1 -20971.97,E2 -20971.97} C_VEL
LIN {X 0,Y 204.327,Z 397.58,A -85,B 0,C 180,E1 -20974.044,E2 -20974.044} C_VEL
LIN {X 0,Y 204.654,Z 396.909,A -85,B 0,C 180,E1 -20977.895,E2 -20977.895} C_VEL
LIN {X 0,Y 205.73,Z 394.647,A -85,B 0,C 180,E1 -20981.827,E2 -20981.827} C_VEL
LIN {X 0,Y 207.034,Z 391.907,A -85,B 0,C 180,E1 -20984.749,E2 -20984.749} C_VEL
LIN {X 0,Y 208.985,Z 388.194,A -85,B 0,C 180,E1 -20987.617,E2 -20987.617} C_VEL
LIN {X 0,Y 211.521,Z 383.423,A -85,B 0,C 180,E1 -20990.418,E2 -20990.418} C_VEL
LIN {X 0,Y 214.584,Z 376.756,A -85,B 0,C 180,E1 -20993.498,E2 -20993.498} C_VEL
LIN {X 0,Y 218.248,Z 368.904,A -85,B 0,C 180,E1 -20996.28,E2 -20996.28} C_VEL
LIN {X 0,Y 222.335,Z 359.577,A -85,B 0,C 180,E1 -20998.819,E2 -20998.819} C_VEL
LIN {X 0,Y 223.755,Z 356.014,A -85,B 0,C 180,E1 -20999.649,E2 -20999.649} C_VEL
LIN {X 0,Y 225.073,Z 346.377,A -85,B 0,C 180,E1 -21002.061,E2 -21002.061} C_VEL
LIN {X 0,Y 225.185,Z 337.608,A -85,B 0,C 180,E1 -21004.178,E2 -21004.178} C_VEL
LIN {X 0,Y 224.359,Z 327.604,A -85,B 0,C 180,E1 -21006.524,E2 -21006.524} C_VEL
LIN {X 0,Y 222.44,Z 317.613,A -85,B 0,C 180,E1 -21008.974,E2 -21008.974} C_VEL
LIN {X 0,Y 220.472,Z 311.464,A -85,B 0,C 180,E1 -21010.64,E2 -21010.64} C_VEL
LIN {X 0,Y 218.338,Z 306.272,A -85,B 0,C 180,E1 -21012.237,E2 -21012.237} C_VEL
LIN {X 0,Y 216.22,Z 302.102,A -85,B 0,C 180,E1 -21013.687,E2 -21013.687} C_VEL
LIN {X 0,Y 215.411,Z 300.674,A -85,B 0,C 180,E1 -21014.21,E2 -21014.21} C_VEL
LIN {X 0,Y 213.327,Z 297.2,A -85,B 0,C 180,E1 -21015.646,E2 -21015.646} C_VEL
LIN {X 0,Y 212.444,Z 295.207,A -85,B 0,C 180,E1 -21016.326,E2 -21016.326} C_VEL
LIN {X 0,Y 209.866,Z 292.081,A -85,B 0,C 180,E1 -21018.031,E2 -21018.031} C_VEL
LIN {X 0,Y 208.673,Z 288.93,A -85,B 0,C 180,E1 -21019.184,E2 -21019.184} C_VEL
LIN {X 0,Y 208.334,Z 286.798,A -85,B 0,C 180,E1 -21024.057,E2 -21024.057} C_VEL
LIN {X 0,Y 208.114,Z 285.534,A -85,B 0,C 180,E1 -21027.589,E2 -21027.589} C_VEL
LIN {X 0,Y 207.982,Z 284.372,A -85,B 0,C 180,E1 -21031.763,E2 -21031.763} C_VEL
LIN {X 0,Y 207.829,Z 283.57,A -85,B 0,C 180,E1 -21036.057,E2 -21036.057} C_VEL
LIN {X 0,Y 207.795,Z 283.08,A -85,B 0,C 180,E1 -21041.26,E2 -21041.26} C_VEL
LIN {X 0,Y 207.912,Z 283.11,A -85,B 0,C 180,E1 -21046.311,E2 -21046.311} C_VEL
LIN {X 0,Y 208.134,Z 283.469,A -85,B 0,C 180,E1 -21050.278,E2 -21050.278} C_VEL
LIN {X 0,Y 208.277,Z 284.138,A -85,B 0,C 180,E1 -21054.188,E2 -21054.188} C_VEL
LIN {X 0,Y 208.473,Z 284.745,A -85,B 0,C 180,E1 -21056.857,E2 -21056.857} C_VEL
LIN {X 0,Y 209.634,Z 287.367,A -85,B 0,C 180,E1 -21057.896,E2 -21057.896} C_VEL
LIN {X 0,Y 212.376,Z 290.2,A -85,B 0,C 180,E1 -21059.737,E2 -21059.737} C_VEL
LIN {X 0,Y 212.883,Z 291.183,A -85,B 0,C 180,E1 -21060.116,E2 -21060.116} C_VEL
LIN {X 0,Y 214.689,Z 294.495,A -85,B 0,C 180,E1 -21061.463,E2 -21061.463} C_VEL
LIN {X 0,Y 215.778,Z 296.053,A -85,B 0,C 180,E1 -21062.179,E2 -21062.179} C_VEL
LIN {X 0,Y 217.937,Z 300.084,A -85,B 0,C 180,E1 -21063.696,E2 -21063.696} C_VEL
LIN {X 0,Y 221.42,Z 307.475,A -85,B 0,C 180,E1 -21066.237,E2 -21066.237} C_VEL
LIN {X 0,Y 223.782,Z 314.405,A -85,B 0,C 180,E1 -21068.275,E2 -21068.275} C_VEL
LIN {X 0,Y 225.874,Z 323.457,A -85,B 0,C 180,E1 -21070.757,E2 -21070.757} C_VEL
LIN {X 0,Y 226.914,Z 331.905,A -85,B 0,C 180,E1 -21072.974,E2 -21072.974} C_VEL
LIN {X 0,Y 227.062,Z 339.903,A -85,B 0,C 180,E1 -21075.1,E2 -21075.1} C_VEL
LIN {X 0,Y 226.946,Z 341.884,A -85,B 0,C 180,E1 -21075.644,E2 -21075.644} C_VEL
LIN {X 0,Y 223.122,Z 351.726,A -85,B 0,C 180,E1 -21077.883,E2 -21077.883} C_VEL
LIN {X 0,Y 219.707,Z 359.513,A -85,B 0,C 180,E1 -21080.11,E2 -21080.11} C_VEL
LIN {X 0,Y 215.896,Z 367.399,A -85,B 0,C 180,E1 -21082.991,E2 -21082.991} C_VEL
LIN {X 0,Y 212.609,Z 373.636,A -85,B 0,C 180,E1 -21085.944,E2 -21085.944} C_VEL
LIN {X 0,Y 209.631,Z 378.995,A -85,B 0,C 180,E1 -21089.35,E2 -21089.35} C_VEL
LIN {X 0,Y 207.398,Z 382.803,A -85,B 0,C 180,E1 -21092.829,E2 -21092.829} C_VEL
LIN {X 0,Y 206.115,Z 384.747,A -85,B 0,C 180,E1 -21095.423,E2 -21095.423} C_VEL
LIN {X 0,Y 205.163,Z 385.96,A -85,B 0,C 180,E1 -21098.065,E2 -21098.065} C_VEL
LIN {X 0,Y 204.455,Z 386.462,A -85,B 0,C 180,E1 -21100.868,E2 -21100.868} C_VEL
LIN {X 0,Y 204.045,Z 386.19,A -85,B 0,C 180,E1 -21103.673,E2 -21103.673} C_VEL
LIN {X 0,Y 203.931,Z 385.167,A -85,B 0,C 180,E1 -21106.43,E2 -21106.43} C_VEL
LIN {X 0,Y 204.039,Z 383.261,A -85,B 0,C 180,E1 -21109.264,E2 -21109.264} C_VEL
LIN {X 0,Y 204.488,Z 380.328,A -85,B 0,C 180,E1 -21112.226,E2 -21112.226} C_VEL
LIN {X 0,Y 205.199,Z 376.21,A -85,B 0,C 180,E1 -21115.28,E2 -21115.28} C_VEL
LIN {X 0,Y 206.236,Z 370.656,A -85,B 0,C 180,E1 -21118.417,E2 -21118.417} C_VEL
LIN {X 0,Y 207.688,Z 363.33,A -85,B 0,C 180,E1 -21121.615,E2 -21121.615} C_VEL
LIN {X 0,Y 209.494,Z 354.887,A -85,B 0,C 180,E1 -21124.525,E2 -21124.525} C_VEL
LIN {X 0,Y 211.289,Z 346.42,A -85,B 0,C 180,E1 -21126.864,E2 -21126.864} C_VEL
LIN {X 0,Y 213.422,Z 335.548,A -85,B 0,C 180,E1 -21129.269,E2 -21129.269} C_VEL
LIN {X 0,Y 214.876,Z 327.848,A -85,B 0,C 180,E1 -21130.661,E2 -21130.661} C_VEL
LIN {X 0,Y 214.138,Z 319.781,A -85,B 0,C 180,E1 -21132.09,E2 -21132.09} C_VEL
LIN {X 0,Y 212.229,Z 307.867,A -85,B 0,C 180,E1 -21133.925,E2 -21133.925} C_VEL
LIN {X 0,Y 209.41,Z 294.202,A -85,B 0,C 180,E1 -21135.67,E2 -21135.67} C_VEL
LIN {X 0,Y 206.157,Z 281.474,A -85,B 0,C 180,E1 -21137.01,E2 -21137.01} C_VEL
LIN {X 0,Y 207.001,Z 277.698,A -85,B 0,C 180,E1 -21142.195,E2 -21142.195} C_VEL
LIN {X 0,Y 207.369,Z 277.653,A -85,B 0,C 180,E1 -21148.058,E2 -21148.058} C_VEL
LIN {X 0,Y 207.51,Z 277.636,A -85,B 0,C 180,E1 -21150,E2 -21150} C_VEL
LIN {X 0,Y 207.376,Z 277.653,A -85,B 0,C 180,E1 -21151.942,E2 -21151.942} C_VEL
LIN {X 0,Y 207.179,Z 277.679,A -85,B 0,C 180,E1 -21157.799,E2 -21157.799} C_VEL
LIN {X 0,Y 206.974,Z 277.701,A -85,B 0,C 180,E1 -21161.756,E2 -21161.756} C_VEL
LIN {X 0,Y 206.859,Z 277.718,A -85,B 0,C 180,E1 -21165.771,E2 -21165.771} C_VEL
LIN {X 0,Y 206.805,Z 277.721,A -85,B 0,C 180,E1 -21169.867,E2 -21169.867} C_VEL
LIN {X 0,Y 206.76,Z 277.729,A -85,B 0,C 180,E1 -21174.072,E2 -21174.072} C_VEL
LIN {X 0,Y 206.728,Z 277.723,A -85,B 0,C 180,E1 -21178.421,E2 -21178.421} C_VEL
LIN {X 0,Y 206.698,Z 277.736,A -85,B 0,C 180,E1 -21182.957,E2 -21182.957} C_VEL
LIN {X 0,Y 206.718,Z 277.731,A -85,B 0,C 180,E1 -21187.731,E2 -21187.731} C_VEL
LIN {X 0,Y 206.742,Z 277.715,A -85,B 0,C 180,E1 -21191.598,E2 -21191.598} C_VEL
LIN {X 0,Y 206.739,Z 277.727,A -85,B 0,C 180,E1 -21195.551,E2 -21195.551} C_VEL
LIN {X 0,Y 206.735,Z 277.733,A -85,B 0,C 180,E1 -21199.77,E2 -21199.77} C_VEL
LIN {X 0,Y 206.725,Z 277.729,A -85,B 0,C 180,E1 -21204.697,E2 -21204.697} C_VEL
LIN {X 0,Y 206.717,Z 277.714,A -85,B 0,C 180,E1 -21209.341,E2 -21209.341} C_VEL
LIN {X 0,Y 206.727,Z 277.727,A -85,B 0,C 180,E1 -21213.774,E2 -21213.774} C_VEL
LIN {X 0,Y 206.752,Z 277.729,A -85,B 0,C 180,E1 -21218.045,E2 -21218.045} C_VEL
LIN {X 0,Y 206.869,Z 277.713,A -85,B 0,C 180,E1 -21222.199,E2 -21222.199} C_VEL
LIN {X 0,Y 206.89,Z 277.696,A -85,B 0,C 180,E1 -21226.246,E2 -21226.246} C_VEL
LIN {X 0,Y 207.096,Z 277.673,A -85,B 0,C 180,E1 -21230.233,E2 -21230.233} C_VEL
LIN {X 0,Y 207.058,Z 277.69,A -85,B 0,C 180,E1 -21234.158,E2 -21234.158} C_VEL
LIN {X 0,Y 207.379,Z 277.654,A -85,B 0,C 180,E1 -21238.06,E2 -21238.06} C_VEL
LIN {X 0,Y 207.512,Z 277.635,A -85,B 0,C 180,E1 -21240.002,E2 -21240.002} C_VEL
LIN {X 0,Y 207.38,Z 277.646,A -85,B 0,C 180,E1 -21241.944,E2 -21241.944} C_VEL
LIN {X 0,Y 207.167,Z 277.671,A -85,B 0,C 180,E1 -21247.801,E2 -21247.801} C_VEL
LIN {X 0,Y 206.98,Z 277.703,A -85,B 0,C 180,E1 -21251.757,E2 -21251.757} C_VEL
LIN {X 0,Y 206.864,Z 277.713,A -85,B 0,C 180,E1 -21255.773,E2 -21255.773} C_VEL
LIN {X 0,Y 206.784,Z 277.72,A -85,B 0,C 180,E1 -21259.871,E2 -21259.871} C_VEL
LIN {X 0,Y 206.765,Z 277.729,A -85,B 0,C 180,E1 -21264.074,E2 -21264.074} C_VEL
LIN {X 0,Y 206.746,Z 277.726,A -85,B 0,C 180,E1 -21268.421,E2 -21268.421} C_VEL
LIN {X 0,Y 206.701,Z 277.739,A -85,B 0,C 180,E1 -21272.96,E2 -21272.96} C_VEL
LIN {X 0,Y 206.683,Z 277.741,A -85,B 0,C 180,E1 -21277.742,E2 -21277.742} C_VEL
LIN {X 0,Y 206.806,Z 277.887,A -85,B 0,C 180,E1 -21283.142,E2 -21283.142} C_VEL
LIN {X 0,Y 207.5,Z 282.037,A -85,B 0,C 180,E1 -21288.174,E2 -21288.174} C_VEL
LIN {X 0,Y 207.953,Z 284.484,A -85,B 0,C 180,E1 -21291.018,E2 -21291.018} C_VEL
LIN {X 0,Y 208.101,Z 285.854,A -85,B 0,C 180,E1 -21292.563,E2 -21292.563} C_VEL
LIN {X 0,Y 207.825,Z 288.029,A -85,B 0,C 180,E1 -21294.909,E2 -21294.909} C_VEL
LIN {X 0,Y 206.825,Z 292.031,A -85,B 0,C 180,E1 -21299.082,E2 -21299.082} C_VEL
LIN {X 0,Y 209.431,Z 305.89,A -85,B 0,C 180,E1 -21300.394,E2 -21300.394} C_VEL
LIN {X 0,Y 211.29,Z 317.614,A -85,B 0,C 180,E1 -21301.794,E2 -21301.794} C_VEL
LIN {X 0,Y 212.543,Z 329.903,A -85,B 0,C 180,E1 -21303.553,E2 -21303.553} C_VEL
LIN {X 0,Y 213.241,Z 340.697,A -85,B 0,C 180,E1 -21305.412,E2 -21305.412} C_VEL
LIN {X 0,Y 213.274,Z 344.727,A -85,B 0,C 180,E1 -21306.192,E2 -21306.192} C_VEL
LIN {X 0,Y 211.262,Z 354.777,A -85,B 0,C 180,E1 -21308.279,E2 -21308.279} C_VEL
LIN {X 0,Y 209.729,Z 361.847,A -85,B 0,C 180,E1 -21310.068,E2 -21310.068} C_VEL
LIN {X 0,Y 208.98,Z 364.561,A -85,B 0,C 180,E1 -21310.822,E2 -21310.822} C_VEL
LIN {X 0,Y 206.907,Z 368.382,A -85,B 0,C 180,E1 -21311.936,E2 -21311.936} C_VEL
LIN {X 0,Y 200.845,Z 376.259,A -85,B 0,C 180,E1 -21314.699,E2 -21314.699} C_VEL
LIN {X 0,Y 199.153,Z 379.358,A -85,B 0,C 180,E1 -21316.071,E2 -21316.071} C_VEL
LIN {X 0,Y 198.889,Z 380.359,A -85,B 0,C 180,E1 -21316.557,E2 -21316.557} C_VEL
LIN {X 0,Y 198.003,Z 386.188,A -85,B 0,C 180,E1 -21319.777,E2 -21319.777} C_VEL
LIN {X 0,Y 197.489,Z 390.471,A -85,B 0,C 180,E1 -21322.845,E2 -21322.845} C_VEL
LIN {X 0,Y 197.253,Z 393.788,A -85,B 0,C 180,E1 -21326.074,E2 -21326.074} C_VEL
LIN {X 0,Y 197.305,Z 395.216,A -85,B 0,C 180,E1 -21327.958,E2 -21327.958} C_VEL
LIN {X 0,Y 197.419,Z 396.363,A -85,B 0,C 180,E1 -21330,E2 -21330} C_VEL
LIN {X 0,Y 197.254,Z 397.338,A -85,B 0,C 180,E1 -21333.929,E2 -21333.929} C_VEL
LIN {X 0,Y 197.348,Z 397.263,A -85,B 0,C 180,E1 -21336.133,E2 -21336.133} C_VEL
LIN {X 0,Y 197.605,Z 396.803,A -85,B 0,C 180,E1 -21338.178,E2 -21338.178} C_VEL
LIN {X 0,Y 198.077,Z 395.938,A -85,B 0,C 180,E1 -21340.218,E2 -21340.218} C_VEL
LIN {X 0,Y 199.627,Z 393.007,A -85,B 0,C 180,E1 -21344.266,E2 -21344.266} C_VEL
LIN {X 0,Y 201.458,Z 389.748,A -85,B 0,C 180,E1 -21347.249,E2 -21347.249} C_VEL
LIN {X 0,Y 203.977,Z 385.479,A -85,B 0,C 180,E1 -21350.154,E2 -21350.154} C_VEL
LIN {X 0,Y 207.148,Z 379.214,A -85,B 0,C 180,E1 -21353.445,E2 -21353.445} C_VEL
LIN {X 0,Y 210.656,Z 372.268,A -85,B 0,C 180,E1 -21356.234,E2 -21356.234} C_VEL
LIN {X 0,Y 214.727,Z 363.805,A -85,B 0,C 180,E1 -21358.865,E2 -21358.865} C_VEL
LIN {X 0,Y 217.656,Z 357.173,A -85,B 0,C 180,E1 -21360.567,E2 -21360.567} C_VEL
LIN {X 0,Y 219.166,Z 347.885,A -85,B 0,C 180,E1 -21363.033,E2 -21363.033} C_VEL
LIN {X 0,Y 219.421,Z 339.43,A -85,B 0,C 180,E1 -21365.206,E2 -21365.206} C_VEL
LIN {X 0,Y 218.898,Z 330.025,A -85,B 0,C 180,E1 -21367.59,E2 -21367.59} C_VEL
LIN {X 0,Y 217.443,Z 321.393,A -85,B 0,C 180,E1 -21369.856,E2 -21369.856} C_VEL
LIN {X 0,Y 215.261,Z 314.202,A -85,B 0,C 180,E1 -21372.047,E2 -21372.047} C_VEL
LIN {X 0,Y 212.129,Z 306.765,A -85,B 0,C 180,E1 -21374.657,E2 -21374.657} C_VEL
LIN {X 0,Y 210.218,Z 303.625,A -85,B 0,C 180,E1 -21376.082,E2 -21376.082} C_VEL
LIN {X 0,Y 209.113,Z 301.06,A -85,B 0,C 180,E1 -21377.062,E2 -21377.062} C_VEL
LIN {X 0,Y 206.808,Z 297.72,A -85,B 0,C 180,E1 -21378.87,E2 -21378.87} C_VEL
LIN {X 0,Y 205.84,Z 295.195,A -85,B 0,C 180,E1 -21379.876,E2 -21379.876} C_VEL
LIN {X 0,Y 202.896,Z 291.966,A -85,B 0,C 180,E1 -21382.369,E2 -21382.369} C_VEL
LIN {X 0,Y 201.567,Z 288.934,A -85,B 0,C 180,E1 -21383.956,E2 -21383.956} C_VEL
LIN {X 0,Y 201.407,Z 288.362,A -85,B 0,C 180,E1 -21384.231,E2 -21384.231} C_VEL
LIN {X 0,Y 201.16,Z 286.965,A -85,B 0,C 180,E1 -21388.393,E2 -21388.393} C_VEL
LIN {X 0,Y 201.008,Z 285.829,A -85,B 0,C 180,E1 -21392.963,E2 -21392.963} C_VEL
LIN {X 0,Y 200.904,Z 285.129,A -85,B 0,C 180,E1 -21397.366,E2 -21397.366} C_VEL
LIN {X 0,Y 200.941,Z 284.777,A -85,B 0,C 180,E1 -21401.65,E2 -21401.65} C_VEL
LIN {X 0,Y 200.984,Z 284.801,A -85,B 0,C 180,E1 -21405.829,E2 -21405.829} C_VEL
LIN {X 0,Y 201.259,Z 285.229,A -85,B 0,C 180,E1 -21410.957,E2 -21410.957} C_VEL
LIN {X 0,Y 201.348,Z 285.574,A -85,B 0,C 180,E1 -21411.909,E2 -21411.909} C_VEL
LIN {X 0,Y 202.547,Z 288.249,A -85,B 0,C 180,E1 -21413.398,E2 -21413.398} C_VEL
LIN {X 0,Y 205.43,Z 290.966,A -85,B 0,C 180,E1 -21415.939,E2 -21415.939} C_VEL
LIN {X 0,Y 206.034,Z 291.771,A -85,B 0,C 180,E1 -21416.453,E2 -21416.453} C_VEL
LIN {X 0,Y 208.013,Z 295.124,A -85,B 0,C 180,E1 -21418.245,E2 -21418.245} C_VEL
LIN {X 0,Y 209.566,Z 296.898,A -85,B 0,C 180,E1 -21419.386,E2 -21419.386} C_VEL
LIN {X 0,Y 211.491,Z 300.614,A -85,B 0,C 180,E1 -21421.009,E2 -21421.009} C_VEL
LIN {X 0,Y 212.565,Z 302.704,A -85,B 0,C 180,E1 -21421.892,E2 -21421.892} C_VEL
LIN {X 0,Y 214.845,Z 307.366,A -85,B 0,C 180,E1 -21423.749,E2 -21423.749} C_VEL
LIN {X 0,Y 217.422,Z 313.597,A -85,B 0,C 180,E1 -21425.994,E2 -21425.994} C_VEL
LIN {X 0,Y 219.778,Z 322.867,A -85,B 0,C 180,E1 -21428.812,E2 -21428.812} C_VEL
LIN {X 0,Y 220.855,Z 330.505,A -85,B 0,C 180,E1 -21431.005,E2 -21431.005} C_VEL
LIN {X 0,Y 221.22,Z 338.662,A -85,B 0,C 180,E1 -21433.314,E2 -21433.314} C_VEL
LIN {X 0,Y 220.951,Z 343.681,A -85,B 0,C 180,E1 -21434.739,E2 -21434.739} C_VEL
LIN {X 0,Y 217.128,Z 352.814,A -85,B 0,C 180,E1 -21436.934,E2 -21436.934} C_VEL
LIN {X 0,Y 212.892,Z 361.747,A -85,B 0,C 180,E1 -21439.674,E2 -21439.674} C_VEL
LIN {X 0,Y 208.867,Z 369.448,A -85,B 0,C 180,E1 -21442.716,E2 -21442.716} C_VEL
LIN {X 0,Y 205.429,Z 375.426,A -85,B 0,C 180,E1 -21445.858,E2 -21445.858} C_VEL
LIN {X 0,Y 202.656,Z 379.947,A -85,B 0,C 180,E1 -21449.043,E2 -21449.043} C_VEL
LIN {X 0,Y 200.337,Z 383.542,A -85,B 0,C 180,E1 -21452.657,E2 -21452.657} C_VEL
LIN {X 0,Y 198.9,Z 385.438,A -85,B 0,C 180,E1 -21455.643,E2 -21455.643} C_VEL
LIN {X 0,Y 197.583,Z 386.648,A -85,B 0,C 180,E1 -21459.807,E2 -21459.807} C_VEL
LIN {X 0,Y 197.05,Z 386.546,A -85,B 0,C 180,E1 -21462.657,E2 -21462.657} C_VEL
LIN {X 0,Y 196.832,Z 385.622,A -85,B 0,C 180,E1 -21465.566,E2 -21465.566} C_VEL
LIN {X 0,Y 196.882,Z 383.846,A -85,B 0,C 180,E1 -21468.554,E2 -21468.554} C_VEL
LIN {X 0,Y 197.266,Z 381.111,A -85,B 0,C 180,E1 -21471.605,E2 -21471.605} C_VEL
LIN {X 0,Y 197.94,Z 377.231,A -85,B 0,C 180,E1 -21474.744,E2 -21474.744} C_VEL
LIN {X 0,Y 198.93,Z 371.923,A -85,B 0,C 180,E1 -21478,E2 -21478} C_VEL
LIN {X 0,Y 200.357,Z 365.051,A -85,B 0,C 180,E1 -21481.269,E2 -21481.269} C_VEL
LIN {X 0,Y 202.145,Z 356.903,A -85,B 0,C 180,E1 -21484.29,E2 -21484.29} C_VEL
LIN {X 0,Y 204.077,Z 347.995,A -85,B 0,C 180,E1 -21486.938,E2 -21486.938} C_VEL
LIN {X 0,Y 206.105,Z 338.198,A -85,B 0,C 180,E1 -21489.282,E2 -21489.282} C_VEL
LIN {X 0,Y 207.98,Z 328.713,A -85,B 0,C 180,E1 -21491.106,E2 -21491.106} C_VEL
LIN {X 0,Y 207.352,Z 321.206,A -85,B 0,C 180,E1 -21492.495,E2 -21492.495} C_VEL
LIN {X 0,Y 205.59,Z 309.711,A -85,B 0,C 180,E1 -21494.384,E2 -21494.384} C_VEL
LIN {X 0,Y 203.258,Z 297.92,A -85,B 0,C 180,E1 -21495.994,E2 -21495.994} C_VEL
LIN {X 0,Y 200.202,Z 285.853,A -85,B 0,C 180,E1 -21497.381,E2 -21497.381} C_VEL
LIN {X 0,Y 199.188,Z 281.666,A -85,B 0,C 180,E1 -21497.843,E2 -21497.843} C_VEL
LIN {X 0,Y 199.933,Z 278.578,A -85,B 0,C 180,E1 -21502.172,E2 -21502.172} C_VEL
LIN {X 0,Y 200.308,Z 278.532,A -85,B 0,C 180,E1 -21507.99,E2 -21507.99} C_VEL
LIN {X 0,Y 200.474,Z 278.512,A -85,B 0,C 180,E1 -21510,E2 -21510} C_VEL
LIN {X 0,Y 200.027,Z 278.569,A -85,B 0,C 180,E1 -21514.03,E2 -21514.03} C_VEL
LIN {X 0,Y 200.123,Z 278.56,A -85,B 0,C 180,E1 -21518.075,E2 -21518.075} C_VEL
LIN {X 0,Y 199.906,Z 278.583,A -85,B 0,C 180,E1 -21522.177,E2 -21522.177} C_VEL
LIN {X 0,Y 199.798,Z 278.594,A -85,B 0,C 180,E1 -21526.344,E2 -21526.344} C_VEL
LIN {X 0,Y 199.734,Z 278.604,A -85,B 0,C 180,E1 -21530.602,E2 -21530.602} C_VEL
LIN {X 0,Y 199.667,Z 278.61,A -85,B 0,C 180,E1 -21534.985,E2 -21534.985} C_VEL
LIN {X 0,Y 199.656,Z 278.605,A -85,B 0,C 180,E1 -21539.525,E2 -21539.525} C_VEL
LIN {X 0,Y 199.65,Z 278.614,A -85,B 0,C 180,E1 -21542.351,E2 -21542.351} C_VEL
LIN {X 0,Y 199.646,Z 278.613,A -85,B 0,C 180,E1 -21546.758,E2 -21546.758} C_VEL
LIN {X 0,Y 199.694,Z 278.601,A -85,B 0,C 180,E1 -21549.308,E2 -21549.308} C_VEL
LIN {X 0,Y 199.683,Z 278.592,A -85,B 0,C 180,E1 -21552.348,E2 -21552.348} C_VEL
LIN {X 0,Y 199.687,Z 278.602,A -85,B 0,C 180,E1 -21555.263,E2 -21555.263} C_VEL
LIN {X 0,Y 199.672,Z 278.611,A -85,B 0,C 180,E1 -21558.033,E2 -21558.033} C_VEL
LIN {X 0,Y 199.695,Z 278.609,A -85,B 0,C 180,E1 -21560.737,E2 -21560.737} C_VEL
LIN {X 0,Y 199.628,Z 278.607,A -85,B 0,C 180,E1 -21565.72,E2 -21565.72} C_VEL
LIN {X 0,Y 199.698,Z 278.589,A -85,B 0,C 180,E1 -21568.14,E2 -21568.14} C_VEL
LIN {X 0,Y 199.681,Z 278.6,A -85,B 0,C 180,E1 -21572.774,E2 -21572.774} C_VEL
LIN {X 0,Y 199.733,Z 278.605,A -85,B 0,C 180,E1 -21577.231,E2 -21577.231} C_VEL
LIN {X 0,Y 199.792,Z 278.593,A -85,B 0,C 180,E1 -21581.76,E2 -21581.76} C_VEL
LIN {X 0,Y 199.83,Z 278.577,A -85,B 0,C 180,E1 -21585.751,E2 -21585.751} C_VEL
LIN {X 0,Y 200.019,Z 278.552,A -85,B 0,C 180,E1 -21589.884,E2 -21589.884} C_VEL
LIN {X 0,Y 200.02,Z 278.566,A -85,B 0,C 180,E1 -21593.952,E2 -21593.952} C_VEL
LIN {X 0,Y 200.318,Z 278.533,A -85,B 0,C 180,E1 -21597.992,E2 -21597.992} C_VEL
LIN {X 0,Y 200.477,Z 278.511,A -85,B 0,C 180,E1 -21600.002,E2 -21600.002} C_VEL
LIN {X 0,Y 200.028,Z 278.551,A -85,B 0,C 180,E1 -21604.032,E2 -21604.032} C_VEL
LIN {X 0,Y 200.11,Z 278.551,A -85,B 0,C 180,E1 -21608.078,E2 -21608.078} C_VEL
LIN {X 0,Y 199.912,Z 278.584,A -85,B 0,C 180,E1 -21612.179,E2 -21612.179} C_VEL
LIN {X 0,Y 199.803,Z 278.589,A -85,B 0,C 180,E1 -21616.346,E2 -21616.346} C_VEL
LIN {X 0,Y 199.7,Z 278.604,A -85,B 0,C 180,E1 -21620.608,E2 -21620.608} C_VEL
LIN {X 0,Y 199.674,Z 278.612,A -85,B 0,C 180,E1 -21624.987,E2 -21624.987} C_VEL
LIN {X 0,Y 199.673,Z 278.611,A -85,B 0,C 180,E1 -21629.525,E2 -21629.525} C_VEL
LIN {X 0,Y 199.674,Z 278.614,A -85,B 0,C 180,E1 -21632.357,E2 -21632.357} C_VEL
LIN {X 0,Y 199.626,Z 278.617,A -85,B 0,C 180,E1 -21636.765,E2 -21636.765} C_VEL
LIN {X 0,Y 199.654,Z 278.616,A -85,B 0,C 180,E1 -21641.978,E2 -21641.978} C_VEL
LIN {X 0,Y 199.725,Z 278.659,A -85,B 0,C 180,E1 -21642.795,E2 -21642.795} C_VEL
LIN {X 0,Y 200.363,Z 282.346,A -85,B 0,C 180,E1 -21647.446,E2 -21647.446} C_VEL
LIN {X 0,Y 200.894,Z 285.263,A -85,B 0,C 180,E1 -21650.972,E2 -21650.972} C_VEL
LIN {X 0,Y 200.966,Z 287.504,A -85,B 0,C 180,E1 -21653.549,E2 -21653.549} C_VEL
LIN {X 0,Y 200.151,Z 291.067,A -85,B 0,C 180,E1 -21657.432,E2 -21657.432} C_VEL
LIN {X 0,Y 199.925,Z 291.972,A -85,B 0,C 180,E1 -21658.306,E2 -21658.306} C_VEL
LIN {X 0,Y 202.447,Z 305.115,A -85,B 0,C 180,E1 -21659.573,E2 -21659.573} C_VEL
LIN {X 0,Y 204.522,Z 318.59,A -85,B 0,C 180,E1 -21661.244,E2 -21661.244} C_VEL
LIN {X 0,Y 205.633,Z 330.276,A -85,B 0,C 180,E1 -21663.002,E2 -21663.002} C_VEL
LIN {X 0,Y 206.312,Z 341.638,A -85,B 0,C 180,E1 -21665.067,E2 -21665.067} C_VEL
LIN {X 0,Y 206.271,Z 345.606,A -85,B 0,C 180,E1 -21665.867,E2 -21665.867} C_VEL
LIN {X 0,Y 204.174,Z 355.498,A -85,B 0,C 180,E1 -21668.041,E2 -21668.041} C_VEL
LIN {X 0,Y 202.481,Z 363.574,A -85,B 0,C 180,E1 -21670.22,E2 -21670.22} C_VEL
LIN {X 0,Y 200.583,Z 372.497,A -85,B 0,C 180,E1 -21673.198,E2 -21673.198} C_VEL
LIN {X 0,Y 199.013,Z 379.66,A -85,B 0,C 180,E1 -21676.21,E2 -21676.21} C_VEL
LIN {X 0,Y 198.889,Z 380.359,A -85,B 0,C 180,E1 -21676.557,E2 -21676.557} C_VEL
LIN {X 0,Y 197.754,Z 383.211,A -85,B 0,C 180,E1 -21678.023,E2 -21678.023} C_VEL
LIN {X 0,Y 194.278,Z 387.218,A -85,B 0,C 180,E1 -21680.473,E2 -21680.473} C_VEL
LIN {X 0,Y 191.518,Z 389.93,A -85,B 0,C 180,E1 -21682.551,E2 -21682.551} C_VEL
LIN {X 0,Y 190.324,Z 391.714,A -85,B 0,C 180,E1 -21684.217,E2 -21684.217} C_VEL
LIN {X 0,Y 190.211,Z 392.262,A -85,B 0,C 180,E1 -21684.79,E2 -21684.79} C_VEL
LIN {X 0,Y 190.21,Z 394.782,A -85,B 0,C 180,E1 -21687.882,E2 -21687.882} C_VEL
LIN {X 0,Y 190.338,Z 395.989,A -85,B 0,C 180,E1 -21690,E2 -21690} C_VEL
LIN {X 0,Y 190.167,Z 397.083,A -85,B 0,C 180,E1 -21693.737,E2 -21693.737} C_VEL
LIN {X 0,Y 190.286,Z 397.083,A -85,B 0,C 180,E1 -21696.361,E2 -21696.361} C_VEL
LIN {X 0,Y 191.071,Z 395.894,A -85,B 0,C 180,E1 -21700.597,E2 -21700.597} C_VEL
LIN {X 0,Y 192.72,Z 393.112,A -85,B 0,C 180,E1 -21704.789,E2 -21704.789} C_VEL
LIN {X 0,Y 194.69,Z 389.972,A -85,B 0,C 180,E1 -21707.868,E2 -21707.868} C_VEL
LIN {X 0,Y 197.346,Z 385.826,A -85,B 0,C 180,E1 -21710.862,E2 -21710.862} C_VEL
LIN {X 0,Y 200.518,Z 379.982,A -85,B 0,C 180,E1 -21714.114,E2 -21714.114} C_VEL
LIN {X 0,Y 204.353,Z 372.963,A -85,B 0,C 180,E1 -21717.108,E2 -21717.108} C_VEL
LIN {X 0,Y 208.599,Z 364.802,A -85,B 0,C 180,E1 -21719.797,E2 -21719.797} C_VEL
LIN {X 0,Y 211.614,Z 358.297,A -85,B 0,C 180,E1 -21721.538,E2 -21721.538} C_VEL
LIN {X 0,Y 213.181,Z 350.085,A -85,B 0,C 180,E1 -21723.851,E2 -21723.851} C_VEL
LIN {X 0,Y 213.728,Z 341.289,A -85,B 0,C 180,E1 -21726.29,E2 -21726.29} C_VEL
LIN {X 0,Y 213.42,Z 332.311,A -85,B 0,C 180,E1 -21728.731,E2 -21728.731} C_VEL
LIN {X 0,Y 212.272,Z 323.984,A -85,B 0,C 180,E1 -21731.127,E2 -21731.127} C_VEL
LIN {X 0,Y 210.466,Z 318.009,A -85,B 0,C 180,E1 -21733.14,E2 -21733.14} C_VEL
LIN {X 0,Y 208.072,Z 311.897,A -85,B 0,C 180,E1 -21735.499,E2 -21735.499} C_VEL
LIN {X 0,Y 205.779,Z 306.969,A -85,B 0,C 180,E1 -21737.658,E2 -21737.658} C_VEL
LIN {X 0,Y 203.917,Z 304.139,A -85,B 0,C 180,E1 -21739.307,E2 -21739.307} C_VEL
LIN {X 0,Y 203.092,Z 301.916,A -85,B 0,C 180,E1 -21740.298,E2 -21740.298} C_VEL
LIN {X 0,Y 199.869,Z 297.19,A -85,B 0,C 180,E1 -21743.625,E2 -21743.625} C_VEL
LIN {X 0,Y 198.927,Z 294.788,A -85,B 0,C 180,E1 -21744.984,E2 -21744.984} C_VEL
LIN {X 0,Y 195.158,Z 290.177,A -85,B 0,C 180,E1 -21750.748,E2 -21750.748} C_VEL
LIN {X 0,Y 194.05,Z 287.185,A -85,B 0,C 180,E1 -21754.879,E2 -21754.879} C_VEL
LIN {X 0,Y 194.002,Z 286.566,A -85,B 0,C 180,E1 -21760.367,E2 -21760.367} C_VEL
LIN {X 0,Y 194.1,Z 286.693,A -85,B 0,C 180,E1 -21761.8,E2 -21761.8} C_VEL
LIN {X 0,Y 197.513,Z 291.153,A -85,B 0,C 180,E1 -21769.447,E2 -21769.447} C_VEL
LIN {X 0,Y 199.13,Z 292.268,A -85,B 0,C 180,E1 -21771.394,E2 -21771.394} C_VEL
LIN {X 0,Y 200.422,Z 295.08,A -85,B 0,C 180,E1 -21773.201,E2 -21773.201} C_VEL
LIN {X 0,Y 203.281,Z 298.345,A -85,B 0,C 180,E1 -21776.033,E2 -21776.033} C_VEL
LIN {X 0,Y 206.327,Z 303.212,A -85,B 0,C 180,E1 -21778.94,E2 -21778.94} C_VEL
LIN {X 0,Y 208.937,Z 308.744,A -85,B 0,C 180,E1 -21781.473,E2 -21781.473} C_VEL
LIN {X 0,Y 211.785,Z 315.351,A -85,B 0,C 180,E1 -21784.236,E2 -21784.236} C_VEL
LIN {X 0,Y 213.353,Z 320.799,A -85,B 0,C 180,E1 -21786.143,E2 -21786.143} C_VEL
LIN {X 0,Y 214.901,Z 329.504,A -85,B 0,C 180,E1 -21788.934,E2 -21788.934} C_VEL
LIN {X 0,Y 215.42,Z 337.188,A -85,B 0,C 180,E1 -21791.286,E2 -21791.286} C_VEL
LIN {X 0,Y 215.026,Z 345.156,A -85,B 0,C 180,E1 -21793.705,E2 -21793.705} C_VEL
LIN {X 0,Y 213.821,Z 348.424,A -85,B 0,C 180,E1 -21794.512,E2 -21794.512} C_VEL
LIN {X 0,Y 210.184,Z 356.118,A -85,B 0,C 180,E1 -21796.561,E2 -21796.561} C_VEL
LIN {X 0,Y 206.225,Z 363.735,A -85,B 0,C 180,E1 -21799.102,E2 -21799.102} C_VEL
LIN {X 0,Y 202.654,Z 369.99,A -85,B 0,C 180,E1 -21801.74,E2 -21801.74} C_VEL
LIN {X 0,Y 198.908,Z 376.066,A -85,B 0,C 180,E1 -21805.084,E2 -21805.084} C_VEL
LIN {X 0,Y 195.591,Z 381.06,A -85,B 0,C 180,E1 -21808.856,E2 -21808.856} C_VEL
LIN {X 0,Y 193.71,Z 383.694,A -85,B 0,C 180,E1 -21811.727,E2 -21811.727} C_VEL
LIN {X 0,Y 191.57,Z 386.181,A -85,B 0,C 180,E1 -21816.189,E2 -21816.189} C_VEL
LIN {X 0,Y 190.61,Z 386.864,A -85,B 0,C 180,E1 -21819.261,E2 -21819.261} C_VEL
LIN {X 0,Y 190.003,Z 386.744,A -85,B 0,C 180,E1 -21822.289,E2 -21822.289} C_VEL
LIN {X 0,Y 189.756,Z 385.807,A -85,B 0,C 180,E1 -21825.277,E2 -21825.277} C_VEL
LIN {X 0,Y 189.764,Z 384.14,A -85,B 0,C 180,E1 -21828.193,E2 -21828.193} C_VEL
LIN {X 0,Y 190.076,Z 381.752,A -85,B 0,C 180,E1 -21831.057,E2 -21831.057} C_VEL
LIN {X 0,Y 190.694,Z 378.212,A -85,B 0,C 180,E1 -21834.17,E2 -21834.17} C_VEL
LIN {X 0,Y 191.65,Z 373.196,A -85,B 0,C 180,E1 -21837.499,E2 -21837.499} C_VEL
LIN {X 0,Y 193.034,Z 366.582,A -85,B 0,C 180,E1 -21840.897,E2 -21840.897} C_VEL
LIN {X 0,Y 194.617,Z 359.602,A -85,B 0,C 180,E1 -21843.747,E2 -21843.747} C_VEL
LIN {X 0,Y 196.756,Z 350.004,A -85,B 0,C 180,E1 -21846.865,E2 -21846.865} C_VEL
LIN {X 0,Y 199.033,Z 339.518,A -85,B 0,C 180,E1 -21849.543,E2 -21849.543} C_VEL
LIN {X 0,Y 201.158,Z 328.98,A -85,B 0,C 180,E1 -21851.674,E2 -21851.674} C_VEL
LIN {X 0,Y 199.986,Z 318.425,A -85,B 0,C 180,E1 -21853.672,E2 -21853.672} C_VEL
LIN {X 0,Y 197.996,Z 306.431,A -85,B 0,C 180,E1 -21855.614,E2 -21855.614} C_VEL
LIN {X 0,Y 195.437,Z 294.216,A -85,B 0,C 180,E1 -21857.276,E2 -21857.276} C_VEL
LIN {X 0,Y 192.245,Z 281.899,A -85,B 0,C 180,E1 -21858.669,E2 -21858.669} C_VEL
LIN {X 0,Y 192.891,Z 279.455,A -85,B 0,C 180,E1 -21862.148,E2 -21862.148} C_VEL
LIN {X 0,Y 193.249,Z 279.412,A -85,B 0,C 180,E1 -21867.916,E2 -21867.916} C_VEL
LIN {X 0,Y 193.437,Z 279.389,A -85,B 0,C 180,E1 -21870,E2 -21870} C_VEL
LIN {X 0,Y 192.973,Z 279.447,A -85,B 0,C 180,E1 -21874.177,E2 -21874.177} C_VEL
LIN {X 0,Y 193.07,Z 279.438,A -85,B 0,C 180,E1 -21878.372,E2 -21878.372} C_VEL
LIN {X 0,Y 192.845,Z 279.464,A -85,B 0,C 180,E1 -21882.631,E2 -21882.631} C_VEL
LIN {X 0,Y 192.773,Z 279.467,A -85,B 0,C 180,E1 -21888.588,E2 -21888.588} C_VEL
LIN {X 0,Y 192.66,Z 279.484,A -85,B 0,C 180,E1 -21894.229,E2 -21894.229} C_VEL
LIN {X 0,Y 192.636,Z 279.477,A -85,B 0,C 180,E1 -21898.89,E2 -21898.89} C_VEL
LIN {X 0,Y 192.59,Z 279.494,A -85,B 0,C 180,E1 -21903.187,E2 -21903.187} C_VEL
LIN {X 0,Y 192.605,Z 279.486,A -85,B 0,C 180,E1 -21908.339,E2 -21908.339} C_VEL
LIN {X 0,Y 192.62,Z 279.473,A -85,B 0,C 180,E1 -21913.141,E2 -21913.141} C_VEL
LIN {X 0,Y 192.614,Z 279.487,A -85,B 0,C 180,E1 -21916.865,E2 -21916.865} C_VEL
LIN {X 0,Y 192.606,Z 279.491,A -85,B 0,C 180,E1 -21921.665,E2 -21921.665} C_VEL
LIN {X 0,Y 192.594,Z 279.479,A -85,B 0,C 180,E1 -21926.817,E2 -21926.817} C_VEL
LIN {X 0,Y 192.659,Z 279.472,A -85,B 0,C 180,E1 -21931.694,E2 -21931.694} C_VEL
LIN {X 0,Y 192.701,Z 279.479,A -85,B 0,C 180,E1 -21936.351,E2 -21936.351} C_VEL
LIN {X 0,Y 192.728,Z 279.473,A -85,B 0,C 180,E1 -21941.46,E2 -21941.46} C_VEL
LIN {X 0,Y 192.758,Z 279.458,A -85,B 0,C 180,E1 -21945.216,E2 -21945.216} C_VEL
LIN {X 0,Y 192.942,Z 279.432,A -85,B 0,C 180,E1 -21949.569,E2 -21949.569} C_VEL
LIN {X 0,Y 192.982,Z 279.441,A -85,B 0,C 180,E1 -21953.73,E2 -21953.73} C_VEL
LIN {X 0,Y 193.26,Z 279.412,A -85,B 0,C 180,E1 -21957.918,E2 -21957.918} C_VEL
LIN {X 0,Y 193.441,Z 279.387,A -85,B 0,C 180,E1 -21960.002,E2 -21960.002} C_VEL
LIN {X 0,Y 192.974,Z 279.428,A -85,B 0,C 180,E1 -21964.179,E2 -21964.179} C_VEL
LIN {X 0,Y 193.061,Z 279.431,A -85,B 0,C 180,E1 -21968.375,E2 -21968.375} C_VEL
LIN {X 0,Y 192.852,Z 279.461,A -85,B 0,C 180,E1 -21972.632,E2 -21972.632} C_VEL
LIN {X 0,Y 192.733,Z 279.465,A -85,B 0,C 180,E1 -21978.544,E2 -21978.544} C_VEL
LIN {X 0,Y 192.666,Z 279.485,A -85,B 0,C 180,E1 -21984.227,E2 -21984.227} C_VEL
LIN {X 0,Y 192.651,Z 279.482,A -85,B 0,C 180,E1 -21988.893,E2 -21988.893} C_VEL
LIN {X 0,Y 192.599,Z 279.497,A -85,B 0,C 180,E1 -21993.188,E2 -21993.188} C_VEL
LIN {X 0,Y 192.556,Z 279.5,A -85,B 0,C 180,E1 -21998.354,E2 -21998.354} C_VEL
LIN {X 0,Y 192.708,Z 279.584,A -85,B 0,C 180,E1 -22002.667,E2 -22002.667} C_VEL
LIN {X 0,Y 193.205,Z 282.652,A -85,B 0,C 180,E1 -22006.682,E2 -22006.682} C_VEL
LIN {X 0,Y 193.644,Z 285.006,A -85,B 0,C 180,E1 -22009.658,E2 -22009.658} C_VEL
LIN {X 0,Y 193.936,Z 287.652,A -85,B 0,C 180,E1 -22012.872,E2 -22012.872} C_VEL
LIN {X 0,Y 193.433,Z 290.159,A -85,B 0,C 180,E1 -22015.727,E2 -22015.727} C_VEL
LIN {X 0,Y 193.052,Z 291.749,A -85,B 0,C 180,E1 -22017.45,E2 -22017.45} C_VEL
LIN {X 0,Y 195.38,Z 304.327,A -85,B 0,C 180,E1 -22018.705,E2 -22018.705} C_VEL
LIN {X 0,Y 197.508,Z 317.855,A -85,B 0,C 180,E1 -22020.444,E2 -22020.444} C_VEL
LIN {X 0,Y 198.701,Z 330.099,A -85,B 0,C 180,E1 -22022.343,E2 -22022.343} C_VEL
LIN {X 0,Y 199.318,Z 341.15,A -85,B 0,C 180,E1 -22024.41,E2 -22024.41} C_VEL
LIN {X 0,Y 199.47,Z 345.203,A -85,B 0,C 180,E1 -22025.267,E2 -22025.267} C_VEL
LIN {X 0,Y 197.209,Z 355.717,A -85,B 0,C 180,E1 -22027.666,E2 -22027.666} C_VEL
LIN {X 0,Y 195.422,Z 364.042,A -85,B 0,C 180,E1 -22030.023,E2 -22030.023} C_VEL
LIN {X 0,Y 193.45,Z 372.837,A -85,B 0,C 180,E1 -22033.104,E2 -22033.104} C_VEL
LIN {X 0,Y 191.836,Z 380.174,A -85,B 0,C 180,E1 -22036.39,E2 -22036.39} C_VEL
LIN {X 0,Y 190.987,Z 385.484,A -85,B 0,C 180,E1 -22039.398,E2 -22039.398} C_VEL
LIN {X 0,Y 190.44,Z 389.877,A -85,B 0,C 180,E1 -22042.579,E2 -22042.579} C_VEL
LIN {X 0,Y 190.211,Z 392.262,A -85,B 0,C 180,E1 -22044.79,E2 -22044.79} C_VEL
LIN {X 0,Y 189.856,Z 393.291,A -85,B 0,C 180,E1 -22045.935,E2 -22045.935} C_VEL
LIN {X 0,Y 188.475,Z 394.553,A -85,B 0,C 180,E1 -22047.642,E2 -22047.642} C_VEL
LIN {X 0,Y 184.165,Z 396.336,A -85,B 0,C 180,E1 -22051.707,E2 -22051.707} C_VEL
LIN {X 0,Y 183.151,Z 396.747,A -85,B 0,C 180,E1 -22053.548,E2 -22053.548} C_VEL
LIN {X 0,Y 183.078,Z 396.845,A -85,B 0,C 180,E1 -22054.172,E2 -22054.172} C_VEL
LIN {X 0,Y 183.219,Z 396.905,A -85,B 0,C 180,E1 -22056.608,E2 -22056.608} C_VEL
LIN {X 0,Y 184.083,Z 395.829,A -85,B 0,C 180,E1 -22061.004,E2 -22061.004} C_VEL
LIN {X 0,Y 184.844,Z 394.731,A -85,B 0,C 180,E1 -22063.186,E2 -22063.186} C_VEL
LIN {X 0,Y 185.833,Z 393.217,A -85,B 0,C 180,E1 -22065.35,E2 -22065.35} C_VEL
LIN {X 0,Y 188.785,Z 388.95,A -85,B 0,C 180,E1 -22069.575,E2 -22069.575} C_VEL
LIN {X 0,Y 191.738,Z 384.605,A -85,B 0,C 180,E1 -22072.635,E2 -22072.635} C_VEL
LIN {X 0,Y 194.897,Z 379.18,A -85,B 0,C 180,E1 -22075.639,E2 -22075.639} C_VEL
LIN {X 0,Y 198.821,Z 372.475,A -85,B 0,C 180,E1 -22078.502,E2 -22078.502} C_VEL
LIN {X 0,Y 203.344,Z 364.232,A -85,B 0,C 180,E1 -22081.226,E2 -22081.226} C_VEL
LIN {X 0,Y 205.627,Z 359.439,A -85,B 0,C 180,E1 -22082.568,E2 -22082.568} C_VEL
LIN {X 0,Y 207.354,Z 351.696,A -85,B 0,C 180,E1 -22084.911,E2 -22084.911} C_VEL
LIN {X 0,Y 208.095,Z 343.16,A -85,B 0,C 180,E1 -22087.438,E2 -22087.438} C_VEL
LIN {X 0,Y 208.03,Z 334.678,A -85,B 0,C 180,E1 -22089.931,E2 -22089.931} C_VEL
LIN {X 0,Y 207.436,Z 328.586,A -85,B 0,C 180,E1 -22091.807,E2 -22091.807} C_VEL
LIN {X 0,Y 205.757,Z 322.092,A -85,B 0,C 180,E1 -22094.166,E2 -22094.166} C_VEL
LIN {X 0,Y 203.822,Z 316.821,A -85,B 0,C 180,E1 -22096.397,E2 -22096.397} C_VEL
LIN {X 0,Y 201.882,Z 312.299,A -85,B 0,C 180,E1 -22098.588,E2 -22098.588} C_VEL
LIN {X 0,Y 199.994,Z 308.269,A -85,B 0,C 180,E1 -22100.76,E2 -22100.76} C_VEL
LIN {X 0,Y 197.042,Z 303.123,A -85,B 0,C 180,E1 -22104.398,E2 -22104.398} C_VEL
LIN {X 0,Y 196.555,Z 301.479,A -85,B 0,C 180,E1 -22105.322,E2 -22105.322} C_VEL
LIN {X 0,Y 192.646,Z 295.339,A -85,B 0,C 180,E1 -22113.16,E2 -22113.16} C_VEL
LIN {X 0,Y 192.376,Z 294.05,A -85,B 0,C 180,E1 -22114.989,E2 -22114.989} C_VEL
LIN {X 0,Y 192.317,Z 293.441,A -85,B 0,C 180,E1 -22120.796,E2 -22120.796} C_VEL
LIN {X 0,Y 192.581,Z 294.191,A -85,B 0,C 180,E1 -22122.749,E2 -22122.749} C_VEL
LIN {X 0,Y 195.484,Z 297.941,A -85,B 0,C 180,E1 -22129.336,E2 -22129.336} C_VEL
LIN {X 0,Y 196.56,Z 298.581,A -85,B 0,C 180,E1 -22130.739,E2 -22130.739} C_VEL
LIN {X 0,Y 197.097,Z 300.221,A -85,B 0,C 180,E1 -22131.798,E2 -22131.798} C_VEL
LIN {X 0,Y 199.604,Z 303.68,A -85,B 0,C 180,E1 -22134.85,E2 -22134.85} C_VEL
LIN {X 0,Y 202.469,Z 308.454,A -85,B 0,C 180,E1 -22138.008,E2 -22138.008} C_VEL
LIN {X 0,Y 204.669,Z 313.362,A -85,B 0,C 180,E1 -22140.52,E2 -22140.52} C_VEL
LIN {X 0,Y 207.449,Z 320.988,A -85,B 0,C 180,E1 -22143.883,E2 -22143.883} C_VEL
LIN {X 0,Y 208.622,Z 326.222,A -85,B 0,C 180,E1 -22145.798,E2 -22145.798} C_VEL
LIN {X 0,Y 209.574,Z 334.238,A -85,B 0,C 180,E1 -22148.556,E2 -22148.556} C_VEL
LIN {X 0,Y 209.56,Z 342.503,A -85,B 0,C 180,E1 -22151.238,E2 -22151.238} C_VEL
LIN {X 0,Y 209.057,Z 347.467,A -85,B 0,C 180,E1 -22152.867,E2 -22152.867} C_VEL
LIN {X 0,Y 205.009,Z 355.759,A -85,B 0,C 180,E1 -22155.079,E2 -22155.079} C_VEL
LIN {X 0,Y 200.727,Z 363.673,A -85,B 0,C 180,E1 -22157.727,E2 -22157.727} C_VEL
LIN {X 0,Y 196.176,Z 371.134,A -85,B 0,C 180,E1 -22160.99,E2 -22160.99} C_VEL
LIN {X 0,Y 192.547,Z 376.591,A -85,B 0,C 180,E1 -22164.149,E2 -22164.149} C_VEL
LIN {X 0,Y 189.654,Z 380.57,A -85,B 0,C 180,E1 -22167.209,E2 -22167.209} C_VEL
LIN {X 0,Y 187.352,Z 383.562,A -85,B 0,C 180,E1 -22170.372,E2 -22170.372} C_VEL
LIN {X 0,Y 185.027,Z 386.163,A -85,B 0,C 180,E1 -22174.73,E2 -22174.73} C_VEL
LIN {X 0,Y 183.93,Z 386.967,A -85,B 0,C 180,E1 -22177.684,E2 -22177.684} C_VEL
LIN {X 0,Y 183.164,Z 387.068,A -85,B 0,C 180,E1 -22180.711,E2 -22180.711} C_VEL
LIN {X 0,Y 182.72,Z 386.431,A -85,B 0,C 180,E1 -22183.811,E2 -22183.811} C_VEL
LIN {X 0,Y 182.64,Z 384.97,A -85,B 0,C 180,E1 -22186.976,E2 -22186.976} C_VEL
LIN {X 0,Y 182.832,Z 382.562,A -85,B 0,C 180,E1 -22190.241,E2 -22190.241} C_VEL
LIN {X 0,Y 183.451,Z 379.12,A -85,B 0,C 180,E1 -22193.558,E2 -22193.558} C_VEL
LIN {X 0,Y 184.349,Z 374.374,A -85,B 0,C 180,E1 -22196.999,E2 -22196.999} C_VEL
LIN {X 0,Y 185.702,Z 368.02,A -85,B 0,C 180,E1 -22200.529,E2 -22200.529} C_VEL
LIN {X 0,Y 187.6,Z 359.905,A -85,B 0,C 180,E1 -22204.033,E2 -22204.033} C_VEL
LIN {X 0,Y 189.413,Z 351.938,A -85,B 0,C 180,E1 -22206.782,E2 -22206.782} C_VEL
LIN {X 0,Y 191.743,Z 341.589,A -85,B 0,C 180,E1 -22209.623,E2 -22209.623} C_VEL
LIN {X 0,Y 194.213,Z 330.148,A -85,B 0,C 180,E1 -22212.087,E2 -22212.087} C_VEL
LIN {X 0,Y 193.39,Z 321.232,A -85,B 0,C 180,E1 -22213.883,E2 -22213.883} C_VEL
LIN {X 0,Y 191.619,Z 309.562,A -85,B 0,C 180,E1 -22215.938,E2 -22215.938} C_VEL
LIN {X 0,Y 189.339,Z 297.8,A -85,B 0,C 180,E1 -22217.677,E2 -22217.677} C_VEL
LIN {X 0,Y 185.813,Z 284.327,A -85,B 0,C 180,E1 -22219.351,E2 -22219.351} C_VEL
LIN {X 0,Y 185.313,Z 282.04,A -85,B 0,C 180,E1 -22219.652,E2 -22219.652} C_VEL
LIN {X 0,Y 185.87,Z 280.328,A -85,B 0,C 180,E1 -22222.396,E2 -22222.396} C_VEL
LIN {X 0,Y 186.191,Z 280.291,A -85,B 0,C 180,E1 -22227.837,E2 -22227.837} C_VEL
LIN {X 0,Y 186.4,Z 280.265,A -85,B 0,C 180,E1 -22230,E2 -22230} C_VEL
LIN {X 0,Y 185.921,Z 280.325,A -85,B 0,C 180,E1 -22234.336,E2 -22234.336} C_VEL
LIN {X 0,Y 186.02,Z 280.314,A -85,B 0,C 180,E1 -22238.692,E2 -22238.692} C_VEL
LIN {X 0,Y 185.756,Z 280.346,A -85,B 0,C 180,E1 -22243.121,E2 -22243.121} C_VEL
LIN {X 0,Y 185.709,Z 280.345,A -85,B 0,C 180,E1 -22247.623,E2 -22247.623} C_VEL
LIN {X 0,Y 185.608,Z 280.366,A -85,B 0,C 180,E1 -22252.25,E2 -22252.25} C_VEL
LIN {X 0,Y 185.553,Z 280.361,A -85,B 0,C 180,E1 -22257.033,E2 -22257.033} C_VEL
LIN {X 0,Y 185.569,Z 280.359,A -85,B 0,C 180,E1 -22259.495,E2 -22259.495} C_VEL
LIN {X 0,Y 185.512,Z 280.376,A -85,B 0,C 180,E1 -22264.629,E2 -22264.629} C_VEL
LIN {X 0,Y 185.56,Z 280.368,A -85,B 0,C 180,E1 -22267.315,E2 -22267.315} C_VEL
LIN {X 0,Y 185.575,Z 280.352,A -85,B 0,C 180,E1 -22270.767,E2 -22270.767} C_VEL
LIN {X 0,Y 185.575,Z 280.363,A -85,B 0,C 180,E1 -22276.017,E2 -22276.017} C_VEL
LIN {X 0,Y 185.554,Z 280.371,A -85,B 0,C 180,E1 -22279.922,E2 -22279.922} C_VEL
LIN {X 0,Y 185.569,Z 280.368,A -85,B 0,C 180,E1 -22282.705,E2 -22282.705} C_VEL
LIN {X 0,Y 185.539,Z 280.351,A -85,B 0,C 180,E1 -22287.977,E2 -22287.977} C_VEL
LIN {X 0,Y 185.576,Z 280.345,A -85,B 0,C 180,E1 -22290.578,E2 -22290.578} C_VEL
LIN {X 0,Y 185.583,Z 280.365,A -85,B 0,C 180,E1 -22295.385,E2 -22295.385} C_VEL
LIN {X 0,Y 185.67,Z 280.353,A -85,B 0,C 180,E1 -22301.136,E2 -22301.136} C_VEL
LIN {X 0,Y 185.69,Z 280.34,A -85,B 0,C 180,E1 -22304.64,E2 -22304.64} C_VEL
LIN {X 0,Y 185.885,Z 280.311,A -85,B 0,C 180,E1 -22309.42,E2 -22309.42} C_VEL
LIN {X 0,Y 185.945,Z 280.317,A -85,B 0,C 180,E1 -22313.492,E2 -22313.492} C_VEL
LIN {X 0,Y 186.204,Z 280.29,A -85,B 0,C 180,E1 -22317.84,E2 -22317.84} C_VEL
LIN {X 0,Y 186.404,Z 280.263,A -85,B 0,C 180,E1 -22320.003,E2 -22320.003} C_VEL
LIN {X 0,Y 185.922,Z 280.305,A -85,B 0,C 180,E1 -22324.338,E2 -22324.338} C_VEL
LIN {X 0,Y 186.008,Z 280.31,A -85,B 0,C 180,E1 -22328.695,E2 -22328.695} C_VEL
LIN {X 0,Y 185.763,Z 280.344,A -85,B 0,C 180,E1 -22333.123,E2 -22333.123} C_VEL
LIN {X 0,Y 185.69,Z 280.343,A -85,B 0,C 180,E1 -22337.627,E2 -22337.627} C_VEL
LIN {X 0,Y 185.598,Z 280.365,A -85,B 0,C 180,E1 -22342.254,E2 -22342.254} C_VEL
LIN {X 0,Y 185.564,Z 280.366,A -85,B 0,C 180,E1 -22347.034,E2 -22347.034} C_VEL
LIN {X 0,Y 185.581,Z 280.365,A -85,B 0,C 180,E1 -22349.495,E2 -22349.495} C_VEL
LIN {X 0,Y 185.501,Z 280.377,A -85,B 0,C 180,E1 -22354.634,E2 -22354.634} C_VEL
LIN {X 0,Y 185.509,Z 280.378,A -85,B 0,C 180,E1 -22357.315,E2 -22357.315} C_VEL
LIN {X 0,Y 185.615,Z 280.382,A -85,B 0,C 180,E1 -22362.348,E2 -22362.348} C_VEL
LIN {X 0,Y 186.219,Z 283.966,A -85,B 0,C 180,E1 -22367.209,E2 -22367.209} C_VEL
LIN {X 0,Y 186.871,Z 287.821,A -85,B 0,C 180,E1 -22372.169,E2 -22372.169} C_VEL
LIN {X 0,Y 186.39,Z 290.649,A -85,B 0,C 180,E1 -22375.557,E2 -22375.557} C_VEL
LIN {X 0,Y 186.161,Z 291.47,A -85,B 0,C 180,E1 -22376.516,E2 -22376.516} C_VEL
LIN {X 0,Y 188.588,Z 304.564,A -85,B 0,C 180,E1 -22377.901,E2 -22377.901} C_VEL
LIN {X 0,Y 190.692,Z 318.419,A -85,B 0,C 180,E1 -22379.781,E2 -22379.781} C_VEL
LIN {X 0,Y 191.842,Z 330.847,A -85,B 0,C 180,E1 -22381.815,E2 -22381.815} C_VEL
LIN {X 0,Y 192.393,Z 341.882,A -85,B 0,C 180,E1 -22384.001,E2 -22384.001} C_VEL
LIN {X 0,Y 192.498,Z 345.86,A -85,B 0,C 180,E1 -22384.886,E2 -22384.886} C_VEL
LIN {X 0,Y 190.034,Z 356.707,A -85,B 0,C 180,E1 -22387.496,E2 -22387.496} C_VEL
LIN {X 0,Y 187.96,Z 366.037,A -85,B 0,C 180,E1 -22390.335,E2 -22390.335} C_VEL
LIN {X 0,Y 186.03,Z 374.346,A -85,B 0,C 180,E1 -22393.54,E2 -22393.54} C_VEL
LIN {X 0,Y 184.59,Z 381.042,A -85,B 0,C 180,E1 -22396.795,E2 -22396.795} C_VEL
LIN {X 0,Y 183.74,Z 386.384,A -85,B 0,C 180,E1 -22400.089,E2 -22400.089} C_VEL
LIN {X 0,Y 183.24,Z 390.515,A -85,B 0,C 180,E1 -22403.393,E2 -22403.393} C_VEL
LIN {X 0,Y 183.089,Z 393.346,A -85,B 0,C 180,E1 -22406.433,E2 -22406.433} C_VEL
LIN {X 0,Y 183.259,Z 395.608,A -85,B 0,C 180,E1 -22410,E2 -22410} C_VEL
LIN {X 0,Y 183.078,Z 396.845,A -85,B 0,C 180,E1 -22414.172,E2 -22414.172} C_VEL
LIN {X 0,Y 182.503,Z 397.007,A -85,B 0,C 180,E1 -22416.013,E2 -22416.013} C_VEL
LIN {X 0,Y 180.068,Z 396.66,A -85,B 0,C 180,E1 -22419.05,E2 -22419.05} C_VEL
LIN {X 0,Y 178.269,Z 395.835,A -85,B 0,C 180,E1 -22421.521,E2 -22421.521} C_VEL
LIN {X 0,Y 177.883,Z 394.899,A -85,B 0,C 180,E1 -22423.404,E2 -22423.404} C_VEL
LIN {X 0,Y 178.053,Z 394.527,A -85,B 0,C 180,E1 -22424.027,E2 -22424.027} C_VEL
LIN {X 0,Y 180.386,Z 391.483,A -85,B 0,C 180,E1 -22428.16,E2 -22428.16} C_VEL
LIN {X 0,Y 183.112,Z 387.957,A -85,B 0,C 180,E1 -22431.383,E2 -22431.383} C_VEL
LIN {X 0,Y 186.231,Z 383.41,A -85,B 0,C 180,E1 -22434.526,E2 -22434.526} C_VEL
LIN {X 0,Y 190.506,Z 376.645,A -85,B 0,C 180,E1 -22438.057,E2 -22438.057} C_VEL
LIN {X 0,Y 194.938,Z 369.449,A -85,B 0,C 180,E1 -22440.913,E2 -22440.913} C_VEL
LIN {X 0,Y 199.748,Z 360.673,A -85,B 0,C 180,E1 -22443.651,E2 -22443.651} C_VEL
LIN {X 0,Y 201.385,Z 354.275,A -85,B 0,C 180,E1 -22445.7,E2 -22445.7} C_VEL
LIN {X 0,Y 202.55,Z 344.989,A -85,B 0,C 180,E1 -22448.648,E2 -22448.648} C_VEL
LIN {X 0,Y 202.705,Z 336.969,A -85,B 0,C 180,E1 -22451.203,E2 -22451.203} C_VEL
LIN {X 0,Y 202.206,Z 331.351,A -85,B 0,C 180,E1 -22453.12,E2 -22453.12} C_VEL
LIN {X 0,Y 201.246,Z 326.937,A -85,B 0,C 180,E1 -22454.875,E2 -22454.875} C_VEL
LIN {X 0,Y 199.447,Z 321.556,A -85,B 0,C 180,E1 -22457.354,E2 -22457.354} C_VEL
LIN {X 0,Y 198.286,Z 318.251,A -85,B 0,C 180,E1 -22459.024,E2 -22459.024} C_VEL
LIN {X 0,Y 196.054,Z 313.183,A -85,B 0,C 180,E1 -22462.057,E2 -22462.057} C_VEL
LIN {X 0,Y 194.269,Z 309.792,A -85,B 0,C 180,E1 -22464.629,E2 -22464.629} C_VEL
LIN {X 0,Y 193.806,Z 308.254,A -85,B 0,C 180,E1 -22465.605,E2 -22465.605} C_VEL
LIN {X 0,Y 190.462,Z 301.814,A -85,B 0,C 180,E1 -22473.715,E2 -22473.715} C_VEL
LIN {X 0,Y 190.222,Z 300.703,A -85,B 0,C 180,E1 -22476.018,E2 -22476.018} C_VEL
LIN {X 0,Y 190.296,Z 300.254,A -85,B 0,C 180,E1 -22480.584,E2 -22480.584} C_VEL
LIN {X 0,Y 190.639,Z 301.44,A -85,B 0,C 180,E1 -22483.431,E2 -22483.431} C_VEL
LIN {X 0,Y 193.955,Z 305.5,A -85,B 0,C 180,E1 -22490.613,E2 -22490.613} C_VEL
LIN {X 0,Y 195.949,Z 309.31,A -85,B 0,C 180,E1 -22493.821,E2 -22493.821} C_VEL
LIN {X 0,Y 197.532,Z 311.92,A -85,B 0,C 180,E1 -22495.917,E2 -22495.917} C_VEL
LIN {X 0,Y 199.132,Z 315.153,A -85,B 0,C 180,E1 -22497.975,E2 -22497.975} C_VEL
LIN {X 0,Y 201.684,Z 322.029,A -85,B 0,C 180,E1 -22501.526,E2 -22501.526} C_VEL
LIN {X 0,Y 203.174,Z 327.528,A -85,B 0,C 180,E1 -22503.965,E2 -22503.965} C_VEL
LIN {X 0,Y 204.042,Z 335.407,A -85,B 0,C 180,E1 -22506.922,E2 -22506.922} C_VEL
LIN {X 0,Y 203.904,Z 343.854,A -85,B 0,C 180,E1 -22509.921,E2 -22509.921} C_VEL
LIN {X 0,Y 203.08,Z 349.814,A -85,B 0,C 180,E1 -22511.982,E2 -22511.982} C_VEL
LIN {X 0,Y 198.588,Z 358.126,A -85,B 0,C 180,E1 -22514.341,E2 -22514.341} C_VEL
LIN {X 0,Y 193.446,Z 366.702,A -85,B 0,C 180,E1 -22517.506,E2 -22517.506} C_VEL
LIN {X 0,Y 189.601,Z 372.453,A -85,B 0,C 180,E1 -22520.276,E2 -22520.276} C_VEL
LIN {X 0,Y 186.217,Z 377.125,A -85,B 0,C 180,E1 -22523.144,E2 -22523.144} C_VEL
LIN {X 0,Y 183.351,Z 380.815,A -85,B 0,C 180,E1 -22526.105,E2 -22526.105} C_VEL
LIN {X 0,Y 180.088,Z 384.608,A -85,B 0,C 180,E1 -22530.483,E2 -22530.483} C_VEL
LIN {X 0,Y 178.157,Z 386.446,A -85,B 0,C 180,E1 -22534.066,E2 -22534.066} C_VEL
LIN {X 0,Y 176.896,Z 387.26,A -85,B 0,C 180,E1 -22537.386,E2 -22537.386} C_VEL
LIN {X 0,Y 176.057,Z 387.227,A -85,B 0,C 180,E1 -22540.673,E2 -22540.673} C_VEL
LIN {X 0,Y 175.608,Z 386.421,A -85,B 0,C 180,E1 -22543.916,E2 -22543.916} C_VEL
LIN {X 0,Y 175.538,Z 384.875,A -85,B 0,C 180,E1 -22547.109,E2 -22547.109} C_VEL
LIN {X 0,Y 175.95,Z 381.264,A -85,B 0,C 180,E1 -22551.651,E2 -22551.651} C_VEL
LIN {X 0,Y 176.62,Z 377.75,A -85,B 0,C 180,E1 -22554.763,E2 -22554.763} C_VEL
LIN {X 0,Y 177.729,Z 372.346,A -85,B 0,C 180,E1 -22558.455,E2 -22558.455} C_VEL
LIN {X 0,Y 179.197,Z 365.819,A -85,B 0,C 180,E1 -22561.926,E2 -22561.926} C_VEL
LIN {X 0,Y 181.157,Z 357.576,A -85,B 0,C 180,E1 -22565.353,E2 -22565.353} C_VEL
LIN {X 0,Y 183.398,Z 348.401,A -85,B 0,C 180,E1 -22568.376,E2 -22568.376} C_VEL
LIN {X 0,Y 185.728,Z 338.073,A -85,B 0,C 180,E1 -22571.076,E2 -22571.076} C_VEL
LIN {X 0,Y 187.388,Z 329.918,A -85,B 0,C 180,E1 -22572.822,E2 -22572.822} C_VEL
LIN {X 0,Y 186.272,Z 319.755,A -85,B 0,C 180,E1 -22574.94,E2 -22574.94} C_VEL
LIN {X 0,Y 184.346,Z 307.803,A -85,B 0,C 180,E1 -22577.058,E2 -22577.058} C_VEL
LIN {X 0,Y 181.864,Z 295.824,A -85,B 0,C 180,E1 -22578.86,E2 -22578.86} C_VEL
LIN {X 0,Y 178.405,Z 282.273,A -85,B 0,C 180,E1 -22580.578,E2 -22580.578} C_VEL
LIN {X 0,Y 178.826,Z 281.205,A -85,B 0,C 180,E1 -22582.378,E2 -22582.378} C_VEL
LIN {X 0,Y 179.136,Z 281.169,A -85,B 0,C 180,E1 -22587.752,E2 -22587.752} C_VEL
LIN {X 0,Y 179.363,Z 281.142,A -85,B 0,C 180,E1 -22590,E2 -22590} C_VEL
LIN {X 0,Y 178.869,Z 281.203,A -85,B 0,C 180,E1 -22594.507,E2 -22594.507} C_VEL
LIN {X 0,Y 178.969,Z 281.191,A -85,B 0,C 180,E1 -22599.037,E2 -22599.037} C_VEL
LIN {X 0,Y 178.68,Z 281.228,A -85,B 0,C 180,E1 -22603.651,E2 -22603.651} C_VEL
LIN {X 0,Y 178.672,Z 281.221,A -85,B 0,C 180,E1 -22608.341,E2 -22608.341} C_VEL
LIN {X 0,Y 178.522,Z 281.247,A -85,B 0,C 180,E1 -22613.183,E2 -22613.183} C_VEL
LIN {X 0,Y 178.478,Z 281.239,A -85,B 0,C 180,E1 -22618.198,E2 -22618.198} C_VEL
LIN {X 0,Y 178.468,Z 281.248,A -85,B 0,C 180,E1 -22620.792,E2 -22620.792} C_VEL
LIN {X 0,Y 178.476,Z 281.253,A -85,B 0,C 180,E1 -22624.22,E2 -22624.22} C_VEL
LIN {X 0,Y 178.478,Z 281.243,A -85,B 0,C 180,E1 -22629.052,E2 -22629.052} C_VEL
LIN {X 0,Y 178.507,Z 281.227,A -85,B 0,C 180,E1 -22632.013,E2 -22632.013} C_VEL
LIN {X 0,Y 178.521,Z 281.236,A -85,B 0,C 180,E1 -22635.122,E2 -22635.122} C_VEL
LIN {X 0,Y 178.506,Z 281.247,A -85,B 0,C 180,E1 -22638.421,E2 -22638.421} C_VEL
LIN {X 0,Y 178.462,Z 281.248,A -85,B 0,C 180,E1 -22643.796,E2 -22643.796} C_VEL
LIN {X 0,Y 178.485,Z 281.236,A -85,B 0,C 180,E1 -22646.55,E2 -22646.55} C_VEL
LIN {X 0,Y 178.517,Z 281.222,A -85,B 0,C 180,E1 -22650.009,E2 -22650.009} C_VEL
LIN {X 0,Y 178.53,Z 281.241,A -85,B 0,C 180,E1 -22654.878,E2 -22654.878} C_VEL
LIN {X 0,Y 178.619,Z 281.233,A -85,B 0,C 180,E1 -22660.787,E2 -22660.787} C_VEL
LIN {X 0,Y 178.653,Z 281.207,A -85,B 0,C 180,E1 -22666.35,E2 -22666.35} C_VEL
LIN {X 0,Y 178.908,Z 281.186,A -85,B 0,C 180,E1 -22670.962,E2 -22670.962} C_VEL
LIN {X 0,Y 179.15,Z 281.169,A -85,B 0,C 180,E1 -22677.754,E2 -22677.754} C_VEL
LIN {X 0,Y 179.368,Z 281.139,A -85,B 0,C 180,E1 -22680.003,E2 -22680.003} C_VEL
LIN {X 0,Y 178.87,Z 281.181,A -85,B 0,C 180,E1 -22684.51,E2 -22684.51} C_VEL
LIN {X 0,Y 178.937,Z 281.19,A -85,B 0,C 180,E1 -22689.042,E2 -22689.042} C_VEL
LIN {X 0,Y 178.686,Z 281.228,A -85,B 0,C 180,E1 -22693.653,E2 -22693.653} C_VEL
LIN {X 0,Y 178.65,Z 281.217,A -85,B 0,C 180,E1 -22698.346,E2 -22698.346} C_VEL
LIN {X 0,Y 178.513,Z 281.248,A -85,B 0,C 180,E1 -22703.187,E2 -22703.187} C_VEL
LIN {X 0,Y 178.489,Z 281.245,A -85,B 0,C 180,E1 -22708.199,E2 -22708.199} C_VEL
LIN {X 0,Y 178.48,Z 281.253,A -85,B 0,C 180,E1 -22710.793,E2 -22710.793} C_VEL
LIN {X 0,Y 178.487,Z 281.251,A -85,B 0,C 180,E1 -22714.221,E2 -22714.221} C_VEL
LIN {X 0,Y 178.412,Z 281.265,A -85,B 0,C 180,E1 -22719.073,E2 -22719.073} C_VEL
LIN {X 0,Y 178.601,Z 281.397,A -85,B 0,C 180,E1 -22722.37,E2 -22722.37} C_VEL
LIN {X 0,Y 179.093,Z 284.37,A -85,B 0,C 180,E1 -22726.554,E2 -22726.554} C_VEL
LIN {X 0,Y 179.726,Z 288.01,A -85,B 0,C 180,E1 -22731.455,E2 -22731.455} C_VEL
LIN {X 0,Y 179.636,Z 290.076,A -85,B 0,C 180,E1 -22734.066,E2 -22734.066} C_VEL
LIN {X 0,Y 179.302,Z 291.314,A -85,B 0,C 180,E1 -22735.573,E2 -22735.573} C_VEL
LIN {X 0,Y 181.84,Z 305.218,A -85,B 0,C 180,E1 -22737.12,E2 -22737.12} C_VEL
LIN {X 0,Y 183.792,Z 318.283,A -85,B 0,C 180,E1 -22738.967,E2 -22738.967} C_VEL
LIN {X 0,Y 184.795,Z 328.306,A -85,B 0,C 180,E1 -22740.652,E2 -22740.652} C_VEL
LIN {X 0,Y 185.423,Z 339.874,A -85,B 0,C 180,E1 -22742.946,E2 -22742.946} C_VEL
LIN {X 0,Y 185.474,Z 346.487,A -85,B 0,C 180,E1 -22744.468,E2 -22744.468} C_VEL
LIN {X 0,Y 182.901,Z 357.494,A -85,B 0,C 180,E1 -22747.256,E2 -22747.256} C_VEL
LIN {X 0,Y 180.838,Z 366.371,A -85,B 0,C 180,E1 -22750.12,E2 -22750.12} C_VEL
LIN {X 0,Y 178.875,Z 374.587,A -85,B 0,C 180,E1 -22753.45,E2 -22753.45} C_VEL
LIN {X 0,Y 177.623,Z 380.191,A -85,B 0,C 180,E1 -22756.267,E2 -22756.267} C_VEL
LIN {X 0,Y 176.736,Z 385.662,A -85,B 0,C 180,E1 -22759.692,E2 -22759.692} C_VEL
LIN {X 0,Y 176.195,Z 389.905,A -85,B 0,C 180,E1 -22763.127,E2 -22763.127} C_VEL
LIN {X 0,Y 176.002,Z 393.143,A -85,B 0,C 180,E1 -22766.68,E2 -22766.68} C_VEL
LIN {X 0,Y 176.181,Z 395.211,A -85,B 0,C 180,E1 -22770,E2 -22770} C_VEL
LIN {X 0,Y 175.999,Z 396.543,A -85,B 0,C 180,E1 -22774.197,E2 -22774.197} C_VEL
LIN {X 0,Y 176.148,Z 396.727,A -85,B 0,C 180,E1 -22776.874,E2 -22776.874} C_VEL
LIN {X 0,Y 177.084,Z 395.763,A -85,B 0,C 180,E1 -22781.445,E2 -22781.445} C_VEL
LIN {X 0,Y 178.053,Z 394.527,A -85,B 0,C 180,E1 -22784.027,E2 -22784.027} C_VEL
LIN {X 0,Y 178.299,Z 393.406,A -85,B 0,C 180,E1 -22785.887,E2 -22785.887} C_VEL
LIN {X 0,Y 177.44,Z 391.125,A -85,B 0,C 180,E1 -22788.985,E2 -22788.985} C_VEL
LIN {X 0,Y 177.007,Z 388.928,A -85,B 0,C 180,E1 -22791.445,E2 -22791.445} C_VEL
LIN {X 0,Y 177.625,Z 386.966,A -85,B 0,C 180,E1 -22793.232,E2 -22793.232} C_VEL
LIN {X 0,Y 178.111,Z 386.224,A -85,B 0,C 180,E1 -22793.8,E2 -22793.8} C_VEL
LIN {X 0,Y 182.243,Z 380.361,A -85,B 0,C 180,E1 -22797.565,E2 -22797.565} C_VEL
LIN {X 0,Y 187.314,Z 372.85,A -85,B 0,C 180,E1 -22801.056,E2 -22801.056} C_VEL
LIN {X 0,Y 192.352,Z 364.844,A -85,B 0,C 180,E1 -22803.861,E2 -22803.861} C_VEL
LIN {X 0,Y 193.899,Z 361.814,A -85,B 0,C 180,E1 -22804.81,E2 -22804.81} C_VEL
LIN {X 0,Y 195.653,Z 355.769,A -85,B 0,C 180,E1 -22806.909,E2 -22806.909} C_VEL
LIN {X 0,Y 197.103,Z 346.871,A -85,B 0,C 180,E1 -22809.926,E2 -22809.926} C_VEL
LIN {X 0,Y 197.457,Z 338.28,A -85,B 0,C 180,E1 -22812.907,E2 -22812.907} C_VEL
LIN {X 0,Y 196.814,Z 332.671,A -85,B 0,C 180,E1 -22815.147,E2 -22815.147} C_VEL
LIN {X 0,Y 195.344,Z 327.104,A -85,B 0,C 180,E1 -22817.837,E2 -22817.837} C_VEL
LIN {X 0,Y 194.438,Z 324.137,A -85,B 0,C 180,E1 -22819.409,E2 -22819.409} C_VEL
LIN {X 0,Y 192.452,Z 318.83,A -85,B 0,C 180,E1 -22822.759,E2 -22822.759} C_VEL
LIN {X 0,Y 190.564,Z 314.151,A -85,B 0,C 180,E1 -22826.411,E2 -22826.411} C_VEL
LIN {X 0,Y 188.016,Z 308.586,A -85,B 0,C 180,E1 -22833.779,E2 -22833.779} C_VEL
LIN {X 0,Y 187.873,Z 307.589,A -85,B 0,C 180,E1 -22835.699,E2 -22835.699} C_VEL
LIN {X 0,Y 187.915,Z 306.955,A -85,B 0,C 180,E1 -22840.328,E2 -22840.328} C_VEL
LIN {X 0,Y 188.083,Z 307.721,A -85,B 0,C 180,E1 -22842.604,E2 -22842.604} C_VEL
LIN {X 0,Y 190.481,Z 311.235,A -85,B 0,C 180,E1 -22849.367,E2 -22849.367} C_VEL
LIN {X 0,Y 191.033,Z 312.153,A -85,B 0,C 180,E1 -22850.468,E2 -22850.468} C_VEL
LIN {X 0,Y 193.525,Z 316.9,A -85,B 0,C 180,E1 -22854.789,E2 -22854.789} C_VEL
LIN {X 0,Y 195.473,Z 321.586,A -85,B 0,C 180,E1 -22857.937,E2 -22857.937} C_VEL
LIN {X 0,Y 197.462,Z 328.289,A -85,B 0,C 180,E1 -22861.528,E2 -22861.528} C_VEL
LIN {X 0,Y 198.301,Z 332.706,A -85,B 0,C 180,E1 -22863.553,E2 -22863.553} C_VEL
LIN {X 0,Y 198.633,Z 340.293,A -85,B 0,C 180,E1 -22866.601,E2 -22866.601} C_VEL
LIN {X 0,Y 198.119,Z 347.084,A -85,B 0,C 180,E1 -22869.183,E2 -22869.183} C_VEL
LIN {X 0,Y 197.415,Z 351.178,A -85,B 0,C 180,E1 -22870.735,E2 -22870.735} C_VEL
LIN {X 0,Y 192.873,Z 359.261,A -85,B 0,C 180,E1 -22873.161,E2 -22873.161} C_VEL
LIN {X 0,Y 187.605,Z 367.484,A -85,B 0,C 180,E1 -22876.314,E2 -22876.314} C_VEL
LIN {X 0,Y 182.803,Z 374.099,A -85,B 0,C 180,E1 -22879.723,E2 -22879.723} C_VEL
LIN {X 0,Y 178.818,Z 379.045,A -85,B 0,C 180,E1 -22883.14,E2 -22883.14} C_VEL
LIN {X 0,Y 176.087,Z 382.181,A -85,B 0,C 180,E1 -22886.039,E2 -22886.039} C_VEL
LIN {X 0,Y 173.821,Z 384.59,A -85,B 0,C 180,E1 -22889.021,E2 -22889.021} C_VEL
LIN {X 0,Y 171.972,Z 386.248,A -85,B 0,C 180,E1 -22892.088,E2 -22892.088} C_VEL
LIN {X 0,Y 170.535,Z 387.249,A -85,B 0,C 180,E1 -22895.233,E2 -22895.233} C_VEL
LIN {X 0,Y 169.447,Z 387.567,A -85,B 0,C 180,E1 -22898.469,E2 -22898.469} C_VEL
LIN {X 0,Y 168.749,Z 387.116,A -85,B 0,C 180,E1 -22901.783,E2 -22901.783} C_VEL
LIN {X 0,Y 168.438,Z 385.901,A -85,B 0,C 180,E1 -22905.175,E2 -22905.175} C_VEL
LIN {X 0,Y 168.5,Z 383.825,A -85,B 0,C 180,E1 -22908.652,E2 -22908.652} C_VEL
LIN {X 0,Y 168.954,Z 380.755,A -85,B 0,C 180,E1 -22912.212,E2 -22912.212} C_VEL
LIN {X 0,Y 169.794,Z 376.487,A -85,B 0,C 180,E1 -22915.87,E2 -22915.87} C_VEL
LIN {X 0,Y 171.018,Z 370.723,A -85,B 0,C 180,E1 -22919.648,E2 -22919.648} C_VEL
LIN {X 0,Y 172.8,Z 363.23,A -85,B 0,C 180,E1 -22923.472,E2 -22923.472} C_VEL
LIN {X 0,Y 174.93,Z 354.759,A -85,B 0,C 180,E1 -22926.846,E2 -22926.846} C_VEL
LIN {X 0,Y 177.024,Z 346.258,A -85,B 0,C 180,E1 -22929.564,E2 -22929.564} C_VEL
LIN {X 0,Y 179.569,Z 335.395,A -85,B 0,C 180,E1 -22932.344,E2 -22932.344} C_VEL
LIN {X 0,Y 180.516,Z 330.89,A -85,B 0,C 180,E1 -22933.314,E2 -22933.314} C_VEL
LIN {X 0,Y 179.254,Z 319.359,A -85,B 0,C 180,E1 -22935.816,E2 -22935.816} C_VEL
LIN {X 0,Y 177.409,Z 307.496,A -85,B 0,C 180,E1 -22937.996,E2 -22937.996} C_VEL
LIN {X 0,Y 174.811,Z 295.411,A -85,B 0,C 180,E1 -22939.91,E2 -22939.91} C_VEL
LIN {X 0,Y 171.557,Z 282.472,A -85,B 0,C 180,E1 -22941.609,E2 -22941.609} C_VEL
LIN {X 0,Y 171.751,Z 282.086,A -85,B 0,C 180,E1 -22942.358,E2 -22942.358} C_VEL
LIN {X 0,Y 172.081,Z 282.048,A -85,B 0,C 180,E1 -22947.66,E2 -22947.66} C_VEL
LIN {X 0,Y 172.325,Z 282.018,A -85,B 0,C 180,E1 -22950,E2 -22950} C_VEL
LIN {X 0,Y 171.818,Z 282.081,A -85,B 0,C 180,E1 -22954.693,E2 -22954.693} C_VEL
LIN {X 0,Y 171.901,Z 282.072,A -85,B 0,C 180,E1 -22959.412,E2 -22959.412} C_VEL
LIN {X 0,Y 171.605,Z 282.111,A -85,B 0,C 180,E1 -22964.225,E2 -22964.225} C_VEL
LIN {X 0,Y 171.567,Z 282.108,A -85,B 0,C 180,E1 -22969.592,E2 -22969.592} C_VEL
LIN {X 0,Y 171.46,Z 282.121,A -85,B 0,C 180,E1 -22975.617,E2 -22975.617} C_VEL
LIN {X 0,Y 171.431,Z 282.125,A -85,B 0,C 180,E1 -22980.587,E2 -22980.587} C_VEL
LIN {X 0,Y 171.399,Z 282.134,A -85,B 0,C 180,E1 -22985.033,E2 -22985.033} C_VEL
LIN {X 0,Y 171.431,Z 282.122,A -85,B 0,C 180,E1 -22988.843,E2 -22988.843} C_VEL
LIN {X 0,Y 171.445,Z 282.116,A -85,B 0,C 180,E1 -22994.176,E2 -22994.176} C_VEL
LIN {X 0,Y 171.423,Z 282.131,A -85,B 0,C 180,E1 -22999.011,E2 -22999.011} C_VEL
LIN {X 0,Y 171.435,Z 282.128,A -85,B 0,C 180,E1 -23002.057,E2 -23002.057} C_VEL
LIN {X 0,Y 171.414,Z 282.109,A -85,B 0,C 180,E1 -23007.795,E2 -23007.795} C_VEL
LIN {X 0,Y 171.443,Z 282.103,A -85,B 0,C 180,E1 -23010.537,E2 -23010.537} C_VEL
LIN {X 0,Y 171.453,Z 282.124,A -85,B 0,C 180,E1 -23015.804,E2 -23015.804} C_VEL
LIN {X 0,Y 171.575,Z 282.11,A -85,B 0,C 180,E1 -23020.874,E2 -23020.874} C_VEL
LIN {X 0,Y 171.571,Z 282.093,A -85,B 0,C 180,E1 -23025.775,E2 -23025.775} C_VEL
LIN {X 0,Y 171.845,Z 282.062,A -85,B 0,C 180,E1 -23030.588,E2 -23030.588} C_VEL
LIN {X 0,Y 171.812,Z 282.081,A -85,B 0,C 180,E1 -23035.31,E2 -23035.31} C_VEL
LIN {X 0,Y 172.331,Z 282.015,A -85,B 0,C 180,E1 -23040.003,E2 -23040.003} C_VEL
LIN {X 0,Y 171.818,Z 282.058,A -85,B 0,C 180,E1 -23044.695,E2 -23044.695} C_VEL
LIN {X 0,Y 171.873,Z 282.07,A -85,B 0,C 180,E1 -23049.416,E2 -23049.416} C_VEL
LIN {X 0,Y 171.608,Z 282.106,A -85,B 0,C 180,E1 -23054.227,E2 -23054.227} C_VEL
LIN {X 0,Y 171.545,Z 282.104,A -85,B 0,C 180,E1 -23059.564,E2 -23059.564} C_VEL
LIN {X 0,Y 171.471,Z 282.124,A -85,B 0,C 180,E1 -23065.619,E2 -23065.619} C_VEL
LIN {X 0,Y 171.443,Z 282.129,A -85,B 0,C 180,E1 -23070.588,E2 -23070.588} C_VEL
LIN {X 0,Y 171.396,Z 282.133,A -85,B 0,C 180,E1 -23075.037,E2 -23075.037} C_VEL
LIN {X 0,Y 171.37,Z 282.141,A -85,B 0,C 180,E1 -23078.813,E2 -23078.813} C_VEL
LIN {X 0,Y 171.526,Z 282.17,A -85,B 0,C 180,E1 -23082.022,E2 -23082.022} C_VEL
LIN {X 0,Y 172.15,Z 285.768,A -85,B 0,C 180,E1 -23087.298,E2 -23087.298} C_VEL
LIN {X 0,Y 172.56,Z 288.219,A -85,B 0,C 180,E1 -23090.703,E2 -23090.703} C_VEL
LIN {X 0,Y 172.621,Z 290.405,A -85,B 0,C 180,E1 -23093.627,E2 -23093.627} C_VEL
LIN {X 0,Y 172.42,Z 291.098,A -85,B 0,C 180,E1 -23094.515,E2 -23094.515} C_VEL
LIN {X 0,Y 174.843,Z 304.092,A -85,B 0,C 180,E1 -23096.05,E2 -23096.05} C_VEL
LIN {X 0,Y 176.684,Z 316.502,A -85,B 0,C 180,E1 -23097.855,E2 -23097.855} C_VEL
LIN {X 0,Y 177.918,Z 328.368,A -85,B 0,C 180,E1 -23099.922,E2 -23099.922} C_VEL
LIN {X 0,Y 178.518,Z 340.528,A -85,B 0,C 180,E1 -23102.446,E2 -23102.446} C_VEL
LIN {X 0,Y 178.449,Z 347.041,A -85,B 0,C 180,E1 -23104.015,E2 -23104.015} C_VEL
LIN {X 0,Y 176.102,Z 356.92,A -85,B 0,C 180,E1 -23106.626,E2 -23106.626} C_VEL
LIN {X 0,Y 174.15,Z 365.123,A -85,B 0,C 180,E1 -23109.322,E2 -23109.322} C_VEL
LIN {X 0,Y 172.067,Z 373.532,A -85,B 0,C 180,E1 -23112.775,E2 -23112.775} C_VEL
LIN {X 0,Y 170.5,Z 380.288,A -85,B 0,C 180,E1 -23116.289,E2 -23116.289} C_VEL
LIN {X 0,Y 169.494,Z 386.496,A -85,B 0,C 180,E1 -23120.453,E2 -23120.453} C_VEL
LIN {X 0,Y 169.035,Z 390.491,A -85,B 0,C 180,E1 -23124.033,E2 -23124.033} C_VEL
LIN {X 0,Y 168.954,Z 393.414,A -85,B 0,C 180,E1 -23127.616,E2 -23127.616} C_VEL
LIN {X 0,Y 169.085,Z 394.808,A -85,B 0,C 180,E1 -23130,E2 -23130} C_VEL
LIN {X 0,Y 168.909,Z 395.943,A -85,B 0,C 180,E1 -23132.995,E2 -23132.995} C_VEL
LIN {X 0,Y 169.1,Z 396.509,A -85,B 0,C 180,E1 -23137.162,E2 -23137.162} C_VEL
LIN {X 0,Y 169.474,Z 396.311,A -85,B 0,C 180,E1 -23139.548,E2 -23139.548} C_VEL
LIN {X 0,Y 171.037,Z 394.691,A -85,B 0,C 180,E1 -23144.357,E2 -23144.357} C_VEL
LIN {X 0,Y 173.663,Z 391.663,A -85,B 0,C 180,E1 -23148.889,E2 -23148.889} C_VEL
LIN {X 0,Y 176.537,Z 388.244,A -85,B 0,C 180,E1 -23152.221,E2 -23152.221} C_VEL
LIN {X 0,Y 178.111,Z 386.224,A -85,B 0,C 180,E1 -23153.8,E2 -23153.8} C_VEL
LIN {X 0,Y 179.215,Z 383.975,A -85,B 0,C 180,E1 -23155.52,E2 -23155.52} C_VEL
LIN {X 0,Y 179.571,Z 380.081,A -85,B 0,C 180,E1 -23158.441,E2 -23158.441} C_VEL
LIN {X 0,Y 180.388,Z 375.62,A -85,B 0,C 180,E1 -23161.236,E2 -23161.236} C_VEL
LIN {X 0,Y 182.137,Z 372.47,A -85,B 0,C 180,E1 -23162.705,E2 -23162.705} C_VEL
LIN {X 0,Y 187.498,Z 364.501,A -85,B 0,C 180,E1 -23165.519,E2 -23165.519} C_VEL
LIN {X 0,Y 189.884,Z 357.712,A -85,B 0,C 180,E1 -23168.012,E2 -23168.012} C_VEL
LIN {X 0,Y 191.431,Z 350.417,A -85,B 0,C 180,E1 -23170.664,E2 -23170.664} C_VEL
LIN {X 0,Y 192.244,Z 343.01,A -85,B 0,C 180,E1 -23173.424,E2 -23173.424} C_VEL
LIN {X 0,Y 192.061,Z 337.979,A -85,B 0,C 180,E1 -23175.512,E2 -23175.512} C_VEL
LIN {X 0,Y 190.915,Z 332.172,A -85,B 0,C 180,E1 -23178.497,E2 -23178.497} C_VEL
LIN {X 0,Y 189.65,Z 327.897,A -85,B 0,C 180,E1 -23181.095,E2 -23181.095} C_VEL
LIN {X 0,Y 188.623,Z 324.491,A -85,B 0,C 180,E1 -23183.402,E2 -23183.402} C_VEL
LIN {X 0,Y 187.17,Z 320.14,A -85,B 0,C 180,E1 -23187.01,E2 -23187.01} C_VEL
LIN {X 0,Y 185.171,Z 314.395,A -85,B 0,C 180,E1 -23195.321,E2 -23195.321} C_VEL
LIN {X 0,Y 185.056,Z 313.755,A -85,B 0,C 180,E1 -23197.678,E2 -23197.678} C_VEL
LIN {X 0,Y 185.2,Z 313.533,A -85,B 0,C 180,E1 -23200.027,E2 -23200.027} C_VEL
LIN {X 0,Y 185.322,Z 314.205,A -85,B 0,C 180,E1 -23202.336,E2 -23202.336} C_VEL
LIN {X 0,Y 187.345,Z 317.594,A -85,B 0,C 180,E1 -23209.187,E2 -23209.187} C_VEL
LIN {X 0,Y 189.929,Z 323.177,A -85,B 0,C 180,E1 -23214.69,E2 -23214.69} C_VEL
LIN {X 0,Y 191.481,Z 327.797,A -85,B 0,C 180,E1 -23217.894,E2 -23217.894} C_VEL
LIN {X 0,Y 192.891,Z 334.356,A -85,B 0,C 180,E1 -23221.565,E2 -23221.565} C_VEL
LIN {X 0,Y 193.23,Z 338.263,A -85,B 0,C 180,E1 -23223.386,E2 -23223.386} C_VEL
LIN {X 0,Y 193.036,Z 344.968,A -85,B 0,C 180,E1 -23226.268,E2 -23226.268} C_VEL
LIN {X 0,Y 192.064,Z 351.439,A -85,B 0,C 180,E1 -23228.902,E2 -23228.902} C_VEL
LIN {X 0,Y 191.75,Z 352.898,A -85,B 0,C 180,E1 -23229.49,E2 -23229.49} C_VEL
LIN {X 0,Y 188.93,Z 357.84,A -85,B 0,C 180,E1 -23231.03,E2 -23231.03} C_VEL
LIN {X 0,Y 183.394,Z 366.094,A -85,B 0,C 180,E1 -23234.087,E2 -23234.087} C_VEL
LIN {X 0,Y 178.944,Z 372.021,A -85,B 0,C 180,E1 -23236.926,E2 -23236.926} C_VEL
LIN {X 0,Y 175.038,Z 376.812,A -85,B 0,C 180,E1 -23239.881,E2 -23239.881} C_VEL
LIN {X 0,Y 170.235,Z 382.093,A -85,B 0,C 180,E1 -23244.38,E2 -23244.38} C_VEL
LIN {X 0,Y 167.227,Z 384.954,A -85,B 0,C 180,E1 -23248.05,E2 -23248.05} C_VEL
LIN {X 0,Y 165.047,Z 386.721,A -85,B 0,C 180,E1 -23251.612,E2 -23251.612} C_VEL
LIN {X 0,Y 163.407,Z 387.618,A -85,B 0,C 180,E1 -23255.2,E2 -23255.2} C_VEL
LIN {X 0,Y 162.241,Z 387.703,A -85,B 0,C 180,E1 -23258.766,E2 -23258.766} C_VEL
LIN {X 0,Y 161.559,Z 387.013,A -85,B 0,C 180,E1 -23262.311,E2 -23262.311} C_VEL
LIN {X 0,Y 161.324,Z 385.567,A -85,B 0,C 180,E1 -23265.812,E2 -23265.812} C_VEL
LIN {X 0,Y 161.436,Z 383.352,A -85,B 0,C 180,E1 -23269.232,E2 -23269.232} C_VEL
LIN {X 0,Y 161.91,Z 380.41,A -85,B 0,C 180,E1 -23272.578,E2 -23272.578} C_VEL
LIN {X 0,Y 162.875,Z 375.683,A -85,B 0,C 180,E1 -23276.623,E2 -23276.623} C_VEL
LIN {X 0,Y 164.256,Z 369.586,A -85,B 0,C 180,E1 -23280.605,E2 -23280.605} C_VEL
LIN {X 0,Y 166.227,Z 361.701,A -85,B 0,C 180,E1 -23284.567,E2 -23284.567} C_VEL
LIN {X 0,Y 168.42,Z 353.169,A -85,B 0,C 180,E1 -23287.942,E2 -23287.942} C_VEL
LIN {X 0,Y 170.896,Z 343.269,A -85,B 0,C 180,E1 -23291.051,E2 -23291.051} C_VEL
LIN {X 0,Y 173.62,Z 331.827,A -85,B 0,C 180,E1 -23293.842,E2 -23293.842} C_VEL
LIN {X 0,Y 172.648,Z 321.805,A -85,B 0,C 180,E1 -23296.164,E2 -23296.164} C_VEL
LIN {X 0,Y 170.992,Z 310.455,A -85,B 0,C 180,E1 -23298.442,E2 -23298.442} C_VEL
LIN {X 0,Y 168.727,Z 298.921,A -85,B 0,C 180,E1 -23300.41,E2 -23300.41} C_VEL
LIN {X 0,Y 165.202,Z 284.802,A -85,B 0,C 180,E1 -23302.438,E2 -23302.438} C_VEL
LIN {X 0,Y 164.751,Z 282.956,A -85,B 0,C 180,E1 -23302.725,E2 -23302.725} C_VEL
LIN {X 0,Y 165.028,Z 282.927,A -85,B 0,C 180,E1 -23307.56,E2 -23307.56} C_VEL
LIN {X 0,Y 165.287,Z 282.895,A -85,B 0,C 180,E1 -23310,E2 -23310} C_VEL
LIN {X 0,Y 164.768,Z 282.959,A -85,B 0,C 180,E1 -23314.894,E2 -23314.894} C_VEL
LIN {X 0,Y 164.844,Z 282.949,A -85,B 0,C 180,E1 -23319.819,E2 -23319.819} C_VEL
LIN {X 0,Y 164.551,Z 282.987,A -85,B 0,C 180,E1 -23324.848,E2 -23324.848} C_VEL
LIN {X 0,Y 164.512,Z 282.989,A -85,B 0,C 180,E1 -23329.984,E2 -23329.984} C_VEL
LIN {X 0,Y 164.385,Z 282.999,A -85,B 0,C 180,E1 -23336.135,E2 -23336.135} C_VEL
LIN {X 0,Y 164.366,Z 283.005,A -85,B 0,C 180,E1 -23341.229,E2 -23341.229} C_VEL
LIN {X 0,Y 164.343,Z 283.011,A -85,B 0,C 180,E1 -23346.776,E2 -23346.776} C_VEL
LIN {X 0,Y 164.368,Z 282.994,A -85,B 0,C 180,E1 -23349.893,E2 -23349.893} C_VEL
LIN {X 0,Y 164.383,Z 282.987,A -85,B 0,C 180,E1 -23353.385,E2 -23353.385} C_VEL
LIN {X 0,Y 164.386,Z 283.002,A -85,B 0,C 180,E1 -23356.844,E2 -23356.844} C_VEL
LIN {X 0,Y 164.369,Z 283.009,A -85,B 0,C 180,E1 -23360.32,E2 -23360.32} C_VEL
LIN {X 0,Y 164.342,Z 283.007,A -85,B 0,C 180,E1 -23364.342,E2 -23364.342} C_VEL
LIN {X 0,Y 164.385,Z 282.978,A -85,B 0,C 180,E1 -23369.137,E2 -23369.137} C_VEL
LIN {X 0,Y 164.411,Z 282.998,A -85,B 0,C 180,E1 -23374.697,E2 -23374.697} C_VEL
LIN {X 0,Y 164.481,Z 282.995,A -85,B 0,C 180,E1 -23380.054,E2 -23380.054} C_VEL
LIN {X 0,Y 164.501,Z 282.975,A -85,B 0,C 180,E1 -23385.15,E2 -23385.15} C_VEL
LIN {X 0,Y 164.765,Z 282.94,A -85,B 0,C 180,E1 -23390.179,E2 -23390.179} C_VEL
LIN {X 0,Y 164.828,Z 282.945,A -85,B 0,C 180,E1 -23392.654,E2 -23392.654} C_VEL
LIN {X 0,Y 165.045,Z 282.925,A -85,B 0,C 180,E1 -23397.562,E2 -23397.562} C_VEL
LIN {X 0,Y 165.293,Z 282.891,A -85,B 0,C 180,E1 -23400.003,E2 -23400.003} C_VEL
LIN {X 0,Y 164.768,Z 282.935,A -85,B 0,C 180,E1 -23404.897,E2 -23404.897} C_VEL
LIN {X 0,Y 164.846,Z 282.938,A -85,B 0,C 180,E1 -23407.351,E2 -23407.351} C_VEL
LIN {X 0,Y 164.751,Z 282.961,A -85,B 0,C 180,E1 -23411.149,E2 -23411.149} C_VEL
LIN {X 0,Y 164.505,Z 282.981,A -85,B 0,C 180,E1 -23417.404,E2 -23417.404} C_VEL
LIN {X 0,Y 164.475,Z 282.987,A -85,B 0,C 180,E1 -23419.992,E2 -23419.992} C_VEL
LIN {X 0,Y 164.396,Z 283.003,A -85,B 0,C 180,E1 -23426.136,E2 -23426.136} C_VEL
LIN {X 0,Y 164.377,Z 283.012,A -85,B 0,C 180,E1 -23431.23,E2 -23431.23} C_VEL
LIN {X 0,Y 164.3,Z 283.018,A -85,B 0,C 180,E1 -23436.791,E2 -23436.791} C_VEL
LIN {X 0,Y 164.476,Z 283.068,A -85,B 0,C 180,E1 -23441.889,E2 -23441.889} C_VEL
LIN {X 0,Y 165.061,Z 286.464,A -85,B 0,C 180,E1 -23447.059,E2 -23447.059} C_VEL
LIN {X 0,Y 165.609,Z 289.915,A -85,B 0,C 180,E1 -23452.024,E2 -23452.024} C_VEL
LIN {X 0,Y 165.571,Z 291.095,A -85,B 0,C 180,E1 -23453.459,E2 -23453.459} C_VEL
LIN {X 0,Y 168.149,Z 304.491,A -85,B 0,C 180,E1 -23455.114,E2 -23455.114} C_VEL
LIN {X 0,Y 169.971,Z 317.719,A -85,B 0,C 180,E1 -23457.154,E2 -23457.154} C_VEL
LIN {X 0,Y 171.113,Z 329.174,A -85,B 0,C 180,E1 -23459.282,E2 -23459.282} C_VEL
LIN {X 0,Y 171.587,Z 339.678,A -85,B 0,C 180,E1 -23461.566,E2 -23461.566} C_VEL
LIN {X 0,Y 171.7,Z 346.335,A -85,B 0,C 180,E1 -23463.24,E2 -23463.24} C_VEL
LIN {X 0,Y 169.371,Z 356.16,A -85,B 0,C 180,E1 -23465.912,E2 -23465.912} C_VEL
LIN {X 0,Y 167.046,Z 365.373,A -85,B 0,C 180,E1 -23469.046,E2 -23469.046} C_VEL
LIN {X 0,Y 164.925,Z 373.682,A -85,B 0,C 180,E1 -23472.645,E2 -23472.645} C_VEL
LIN {X 0,Y 163.367,Z 380.377,A -85,B 0,C 180,E1 -23476.313,E2 -23476.313} C_VEL
LIN {X 0,Y 162.482,Z 385.723,A -85,B 0,C 180,E1 -23480.037,E2 -23480.037} C_VEL
LIN {X 0,Y 161.969,Z 389.851,A -85,B 0,C 180,E1 -23483.772,E2 -23483.772} C_VEL
LIN {X 0,Y 161.872,Z 392.895,A -85,B 0,C 180,E1 -23487.511,E2 -23487.511} C_VEL
LIN {X 0,Y 161.992,Z 394.386,A -85,B 0,C 180,E1 -23490,E2 -23490} C_VEL
LIN {X 0,Y 161.84,Z 395.486,A -85,B 0,C 180,E1 -23492.768,E2 -23492.768} C_VEL
LIN {X 0,Y 162.032,Z 396.272,A -85,B 0,C 180,E1 -23497.476,E2 -23497.476} C_VEL
LIN {X 0,Y 163.154,Z 395.653,A -85,B 0,C 180,E1 -23502.437,E2 -23502.437} C_VEL
LIN {X 0,Y 165.312,Z 393.468,A -85,B 0,C 180,E1 -23507.313,E2 -23507.313} C_VEL
LIN {X 0,Y 168.903,Z 389.77,A -85,B 0,C 180,E1 -23511.992,E2 -23511.992} C_VEL
LIN {X 0,Y 172.274,Z 385.864,A -85,B 0,C 180,E1 -23515.362,E2 -23515.362} C_VEL
LIN {X 0,Y 176.008,Z 380.937,A -85,B 0,C 180,E1 -23518.629,E2 -23518.629} C_VEL
LIN {X 0,Y 181.326,Z 373.672,A -85,B 0,C 180,E1 -23522.203,E2 -23522.203} C_VEL
LIN {X 0,Y 182.137,Z 372.47,A -85,B 0,C 180,E1 -23522.705,E2 -23522.705} C_VEL
LIN {X 0,Y 183.918,Z 369.189,A -85,B 0,C 180,E1 -23524.139,E2 -23524.139} C_VEL
LIN {X 0,Y 184.668,Z 366.046,A -85,B 0,C 180,E1 -23525.697,E2 -23525.697} C_VEL
LIN {X 0,Y 184.867,Z 359.775,A -85,B 0,C 180,E1 -23528.927,E2 -23528.927} C_VEL
LIN {X 0,Y 185.443,Z 355.091,A -85,B 0,C 180,E1 -23530.981,E2 -23530.981} C_VEL
LIN {X 0,Y 186.748,Z 348.043,A -85,B 0,C 180,E1 -23533.77,E2 -23533.77} C_VEL
LIN {X 0,Y 187.089,Z 343.836,A -85,B 0,C 180,E1 -23535.538,E2 -23535.538} C_VEL
LIN {X 0,Y 186.612,Z 338.765,A -85,B 0,C 180,E1 -23538.174,E2 -23538.174} C_VEL
LIN {X 0,Y 185.641,Z 334.034,A -85,B 0,C 180,E1 -23541.085,E2 -23541.085} C_VEL
LIN {X 0,Y 184.663,Z 330.219,A -85,B 0,C 180,E1 -23543.845,E2 -23543.845} C_VEL
LIN {X 0,Y 183.526,Z 326.012,A -85,B 0,C 180,E1 -23547.577,E2 -23547.577} C_VEL
LIN {X 0,Y 182.077,Z 321.163,A -85,B 0,C 180,E1 -23554.873,E2 -23554.873} C_VEL
LIN {X 0,Y 182.05,Z 320.153,A -85,B 0,C 180,E1 -23557.894,E2 -23557.894} C_VEL
LIN {X 0,Y 182.147,Z 319.997,A -85,B 0,C 180,E1 -23559.678,E2 -23559.678} C_VEL
LIN {X 0,Y 182.239,Z 320.505,A -85,B 0,C 180,E1 -23562.027,E2 -23562.027} C_VEL
LIN {X 0,Y 183.879,Z 323.79,A -85,B 0,C 180,E1 -23568.98,E2 -23568.98} C_VEL
LIN {X 0,Y 186.014,Z 329.192,A -85,B 0,C 180,E1 -23574.577,E2 -23574.577} C_VEL
LIN {X 0,Y 187.115,Z 333.788,A -85,B 0,C 180,E1 -23577.845,E2 -23577.845} C_VEL
LIN {X 0,Y 187.945,Z 339.197,A -85,B 0,C 180,E1 -23581.072,E2 -23581.072} C_VEL
LIN {X 0,Y 187.887,Z 344.678,A -85,B 0,C 180,E1 -23583.751,E2 -23583.751} C_VEL
LIN {X 0,Y 187.041,Z 350.733,A -85,B 0,C 180,E1 -23586.47,E2 -23586.47} C_VEL
LIN {X 0,Y 186.163,Z 354.499,A -85,B 0,C 180,E1 -23588.136,E2 -23588.136} C_VEL
LIN {X 0,Y 184.993,Z 356.871,A -85,B 0,C 180,E1 -23588.985,E2 -23588.985} C_VEL
LIN {X 0,Y 179.478,Z 364.804,A -85,B 0,C 180,E1 -23591.784,E2 -23591.784} C_VEL
LIN {X 0,Y 174.426,Z 371.248,A -85,B 0,C 180,E1 -23594.763,E2 -23594.763} C_VEL
LIN {X 0,Y 168.985,Z 377.461,A -85,B 0,C 180,E1 -23598.648,E2 -23598.648} C_VEL
LIN {X 0,Y 164.524,Z 381.991,A -85,B 0,C 180,E1 -23602.606,E2 -23602.606} C_VEL
LIN {X 0,Y 161.681,Z 384.523,A -85,B 0,C 180,E1 -23605.762,E2 -23605.762} C_VEL
LIN {X 0,Y 159.313,Z 386.369,A -85,B 0,C 180,E1 -23609.026,E2 -23609.026} C_VEL
LIN {X 0,Y 157.438,Z 387.521,A -85,B 0,C 180,E1 -23612.386,E2 -23612.386} C_VEL
LIN {X 0,Y 156.003,Z 387.97,A -85,B 0,C 180,E1 -23615.845,E2 -23615.845} C_VEL
LIN {X 0,Y 154.93,Z 387.717,A -85,B 0,C 180,E1 -23619.544,E2 -23619.544} C_VEL
LIN {X 0,Y 154.364,Z 386.693,A -85,B 0,C 180,E1 -23623.244,E2 -23623.244} C_VEL
LIN {X 0,Y 154.222,Z 384.881,A -85,B 0,C 180,E1 -23626.879,E2 -23626.879} C_VEL
LIN {X 0,Y 154.486,Z 382.162,A -85,B 0,C 180,E1 -23630.653,E2 -23630.653} C_VEL
LIN {X 0,Y 155.242,Z 378.332,A -85,B 0,C 180,E1 -23634.57,E2 -23634.57} C_VEL
LIN {X 0,Y 156.368,Z 373.111,A -85,B 0,C 180,E1 -23638.638,E2 -23638.638} C_VEL
LIN {X 0,Y 158.061,Z 366.259,A -85,B 0,C 180,E1 -23642.775,E2 -23642.775} C_VEL
LIN {X 0,Y 160.338,Z 357.68,A -85,B 0,C 180,E1 -23646.767,E2 -23646.767} C_VEL
